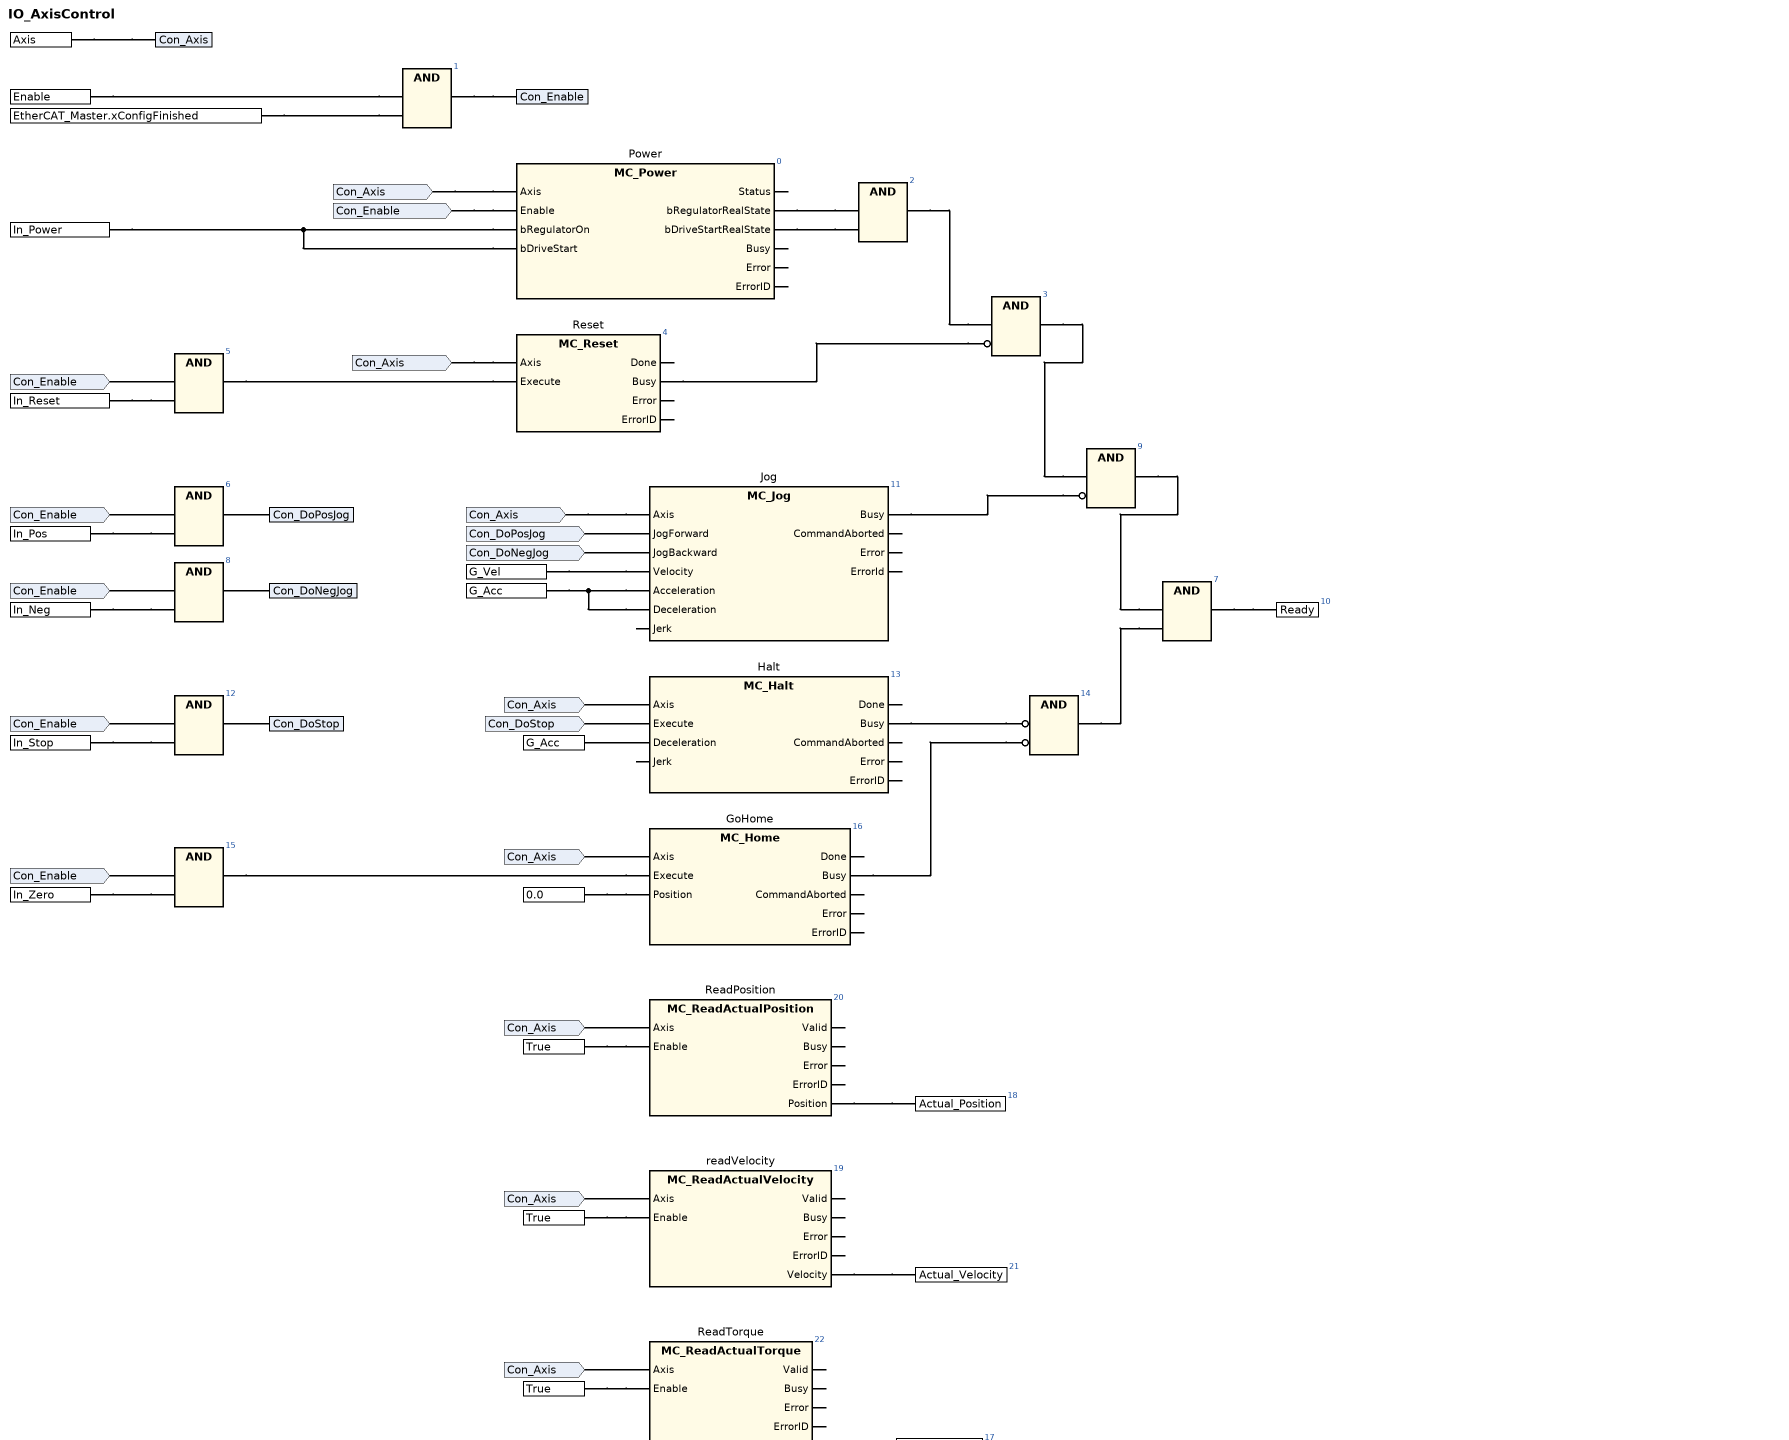
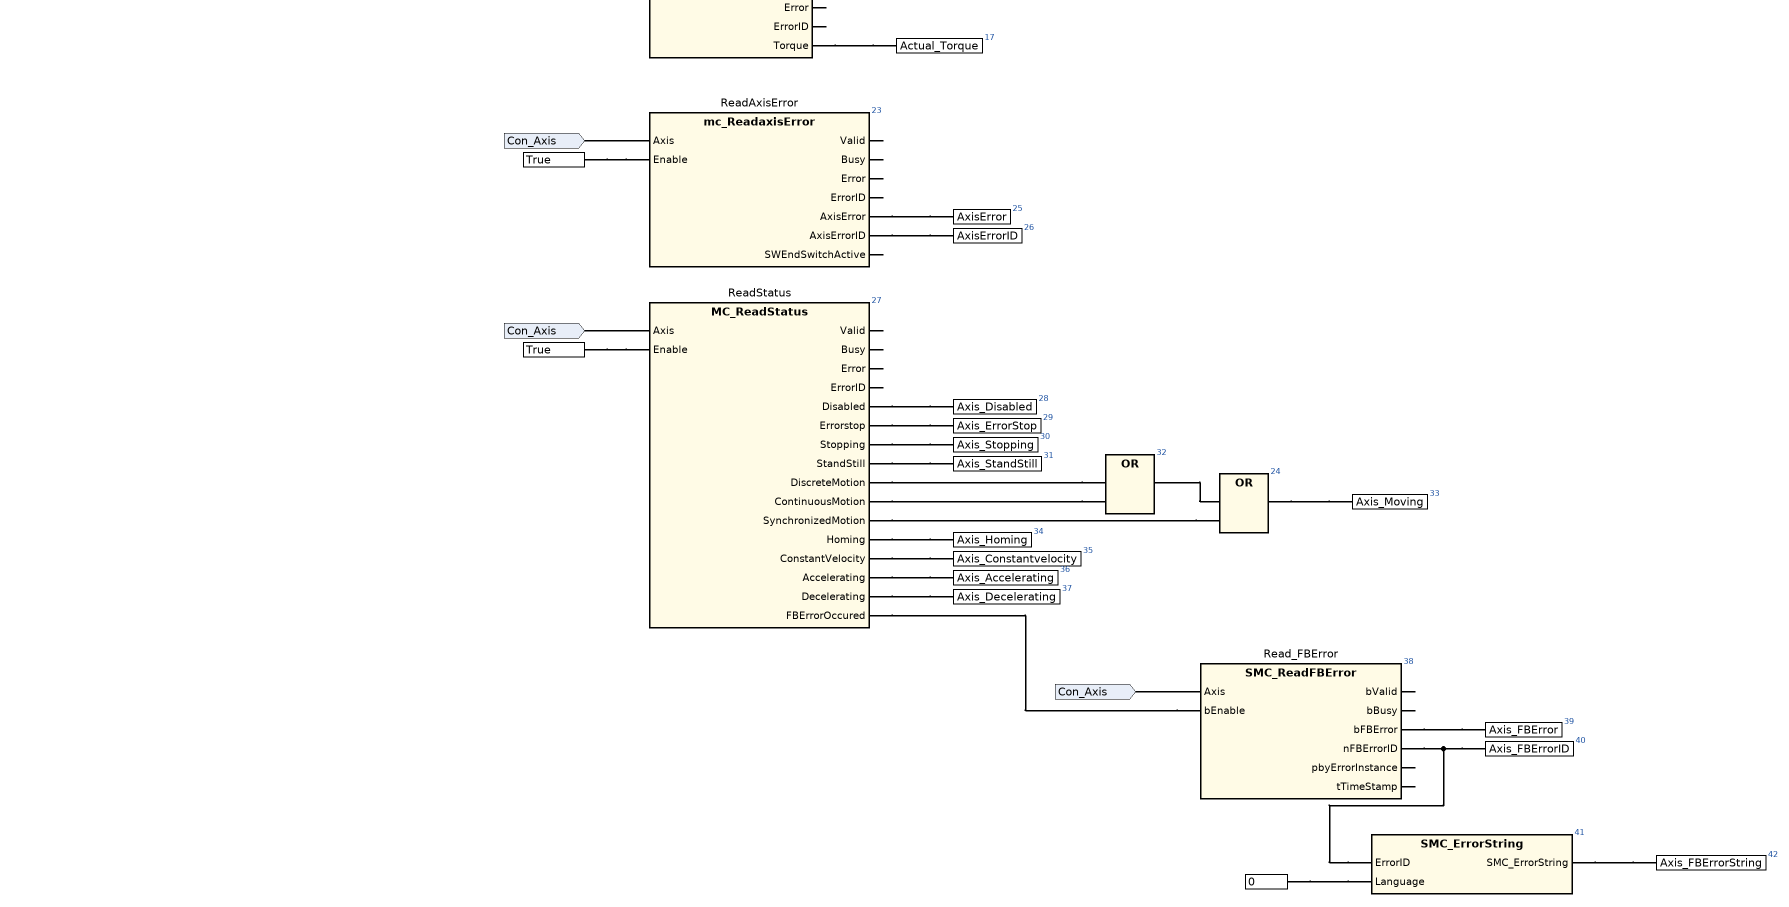
Power(Axis := _w1, Enable := _w2, bRegulatorOn := In_Power, bDriveStart := In_Power); // MC_Power
(* Enable AND EtherCAT_Master.xConfigFinished; result not used *)
_w3 := (Power.bRegulatorRealState AND Power.bDriveStartRealState) AND NOT Reset.Busy;
Reset(Axis := _w4, Execute := _w5); // MC_Reset
_w5 := _w6 AND In_Reset;
(* _w7 AND In_Pos; result not used *)
_w10 := _w8 AND _w9;
(* _w11 AND In_Neg; result not used *)
_w8 := _w3 AND NOT Jog.Busy;
Ready := _w10;
Jog(
    Axis := _w12,
    JogForward := _w13,
    JogBackward := _w14,
    Velocity := G_Vel,
    Acceleration := G_Acc,
    Deceleration := G_Acc); // MC_Jog
(* _w15 AND In_Stop; result not used *)
Halt(Axis := _w16, Execute := _w17, Deceleration := G_Acc); // MC_Halt
_w9 := NOT Halt.Busy AND NOT GoHome.Busy;
GoHome(Axis := _w19, Execute := _w18 AND In_Zero, Position := 0.0); // MC_Home
Actual_Torque := ReadTorque.Torque;
Actual_Position := ReadPosition.Position;
readVelocity(Axis := _w20, Enable := True); // MC_ReadActualVelocity
ReadPosition(Axis := _w21, Enable := True); // MC_ReadActualPosition
Actual_Velocity := readVelocity.Velocity;
ReadTorque(Axis := _w22, Enable := True); // MC_ReadActualTorque
ReadAxisError(Axis := _w23, Enable := True); // mc_ReadaxisError
_w25 := _w24 OR ReadStatus.SynchronizedMotion;
AxisError := ReadAxisError.AxisError;
AxisErrorID := ReadAxisError.AxisErrorID;
ReadStatus(Axis := _w26, Enable := True); // MC_ReadStatus
Axis_Disabled := ReadStatus.Disabled;
Axis_ErrorStop := ReadStatus.Errorstop;
Axis_Stopping := ReadStatus.Stopping;
Axis_StandStill := ReadStatus.StandStill;
_w24 := ReadStatus.DiscreteMotion OR ReadStatus.ContinuousMotion;
Axis_Moving := _w25;
Axis_Homing := ReadStatus.Homing;
Axis_Constantvelocity := ReadStatus.ConstantVelocity;
Axis_Accelerating := ReadStatus.Accelerating;
Axis_Decelerating := ReadStatus.Decelerating;
Read_FBError(Axis := _w27, bEnable := ReadStatus.FBErrorOccured); // SMC_ReadFBError
Axis_FBError := Read_FBError.bFBError;
Axis_FBErrorID := Read_FBError.nFBErrorID;
_w28 := SMC_ErrorString(ErrorID := Read_FBError.nFBErrorID, Language := 0);
Axis_FBErrorString := _w28;

END_FUNCTION_BLOCK

// LogHiCycleCount
PROGRAM LogHiCycleCount
VAR
	strMsg: STRING[255];
	iStatus : INT := 0;
	LogIndex :DINT := 0;
	LogMsg : ARRAY [1..200] OF STRING[255];
	LogType : STRING;
	
	CycleTimeWarning: DWORD := 600;
	TotalSyncBufferAvgWarning: DINT := 125;
	CycleTimeError: DWORD := 900;
	TotalSyncBufferAvgError: DINT := 200;
END_VAR

VAR_INPUT
	bResetArray: BOOL;
END_VAR


IF bResetArray = TRUE THEN
	LogIndex := 0;
END_IF




CASE iStatus OF
	
0:	//Wait for Distributed Clocks in sync
	IF GVL.DC_InSync THEN
		iStatus:=iStatus + 1;
	END_IF
1: 	//Wait for High Cycle Count
	LogType := 'None';
	IF (DC_Monitor.CycleTime_Last > CycleTimeWarning OR DC_Monitor.TotalSyncBufferAvg > TotalSyncBufferAvgWarning) THEN
		iStatus := iStatus + 1;
	END_IF

2:	//Log Data
	LogIndex := LogIndex + 1;
	IF (DC_Monitor.CycleTime_Last > CycleTimeError OR DC_Monitor.TotalSyncBufferAvg > TotalSyncBufferAvgError) THEN
		LogType := 'Error';
	ELSE
		LogType := 'Warning';
	END_IF
	LogMsg[LogIndex] :=  GetLogMsgString();
	
	iStatus := 2;

END_CASE

END_PROGRAM

// GetLogMsgString
FUNCTION GetLogMsgString : STRING[255]
VAR_INPUT
END_VAR
VAR
	msg: STRING[255];
	seperator: STRING;
	eol:String;
	
	strTemp0: STRING[255];
	strTemp1: STRING[255];
END_VAR

eol := WORD_AS_STRING(16#0A0D, FALSE);
seperator := ',';

(*
strTemp0 := Concat(Concat(Concat(Concat(Concat(Concat(Concat(Concat(Concat(Concat(Concat(Concat(Concat(Concat(	My_FLOAT_TO_STRING(X.fSetPosition), 
																												seperator), 
																												My_FLOAT_TO_STRING(Y.fSetPosition)),  
																												seperator), 
																												My_FLOAT_TO_STRING(Z.fSetPosition)),  
																												seperator), 
																												My_FLOAT_TO_STRING(BB.fSetPosition)),  
																												seperator), 
																												My_FLOAT_TO_STRING(CC.fSetPosition)),  
																												seperator), 
																												My_FLOAT_TO_STRING(GGX.fSetPosition)),  
																												seperator), 
																												My_FLOAT_TO_STRING(GGZ.fSetPosition)),  
																												seperator), 
																												My_FLOAT_TO_STRING(GGC.fSetPosition));
																												
strTemp1 := Concat(Concat(Concat(Concat(Concat(Concat(Concat(Concat(Concat(Concat(Concat(Concat(Concat(Concat(	My_FLOAT_TO_STRING(X.fActPosition), 
																												seperator), 
																												My_FLOAT_TO_STRING(Y.fActPosition)),  
																												seperator), 
																												My_FLOAT_TO_STRING(Z.fActPosition)),  
																												seperator), 
																												My_FLOAT_TO_STRING(BB.fActPosition)),  
																												seperator), 
																												My_FLOAT_TO_STRING(CC.fActPosition)),  
																												seperator), 
																												My_FLOAT_TO_STRING(GGX.fActPosition)),  
																												seperator), 
																												My_FLOAT_TO_STRING(GGZ.fActPosition)),  
																												seperator), 
																												My_FLOAT_TO_STRING(GGC.fActPosition));
*)


strTemp0 := My_FLOAT_TO_STRING();
strTemp1 := 'TotalSyncBufferAvg';
GetLogMsgString := Concat(Concat(Concat(Concat(Concat(	GetTimeStampString(),
														seperator),
														strTemp0), 
														seperator),
														strTemp1), 
														eol);

END_FUNCTION

// My_FLOAT_TO_STRING
FUNCTION My_FLOAT_TO_STRING : STRING(10)
VAR_INPUT
	Value : LREAL;
END_VAR
VAR
	intTemp : DINT;
END_VAR

//My_LREAL_TO_STRING := REAL_TO_STRING(Value);
intTemp := LREAL_TO_DINT(Value * 1000);
My_FLOAT_TO_STRING := LREAL_TO_STRING(DINT_TO_LREAL(intTemp)/1000 );

END_FUNCTION

// GetTimeStampString
FUNCTION GetTimeStampString : String
VAR_INPUT
END_VAR
VAR
	TimeStamp : SysTime;
	StructTimeStamp : SysTimeDate;
	Result : RTS_IEC_RESULT;
	StrDate : STRING;
	StrTime : STRING;
	
END_VAR

Result := systimertc.SysTimeRtcHighResGet(pTimestamp := TimeStamp);

Result := systimertc.SysTimeRtcConvertHighResToLocal(pTimeStamp:=TimeStamp, pDate:=StructTimeStamp);

StrDate := UINT_TO_STRING(StructTimeStamp.wYear);
IF StructTimeStamp.wMonth < 10 THEN 
	StrDate := Concat(Concat(StrDate, '0') , UINT_TO_STRING(StructTimeStamp.wMonth));
ELSE
	StrDate := Concat(StrDate , UINT_TO_STRING(StructTimeStamp.wMonth));
END_IF

IF StructTimeStamp.wDay < 10 THEN 
	StrDate := Concat(Concat(StrDate , '0') , UINT_TO_STRING(StructTimeStamp.wDay));
ELSE
	StrDate := Concat(StrDate , UINT_TO_STRING(StructTimeStamp.wDay));
END_IF


IF StructTimeStamp.wHour < 10 THEN 
	StrTime := Concat(Concat('0' , UINT_TO_STRING(StructTimeStamp.wHour)) , ':');
ELSE
	StrTime := Concat(UINT_TO_STRING(StructTimeStamp.wHour) , ':');
END_IF

IF StructTimeStamp.wMinute < 10 THEN 
	StrTime := Concat(Concat(Concat(StrTime , '0') , UINT_TO_STRING(StructTimeStamp.wMinute)), ':');
ELSE
	StrTime := Concat(Concat(StrTime , UINT_TO_STRING(StructTimeStamp.wMinute)), ':');
END_IF

IF StructTimeStamp.wSecond < 10 THEN 
	StrTime := Concat(Concat(Concat(StrTime , '0') , UINT_TO_STRING(StructTimeStamp.wSecond)) , '.');
ELSE
	StrTime := Concat(Concat(StrTime , UINT_TO_STRING(StructTimeStamp.wSecond)) , '.');
END_IF

IF StructTimeStamp.wMilliseconds < 10 THEN 
	StrTime := Concat(Concat(StrTime , '00') , UINT_TO_STRING(StructTimeStamp.wMilliseconds));
ELSE
	IF StructTimeStamp.wMilliseconds < 100 THEN 
		StrTime := Concat(Concat(StrTime , '0') , UINT_TO_STRING(StructTimeStamp.wMilliseconds));
	ELSE
		StrTime := Concat(StrTime , UINT_TO_STRING(StructTimeStamp.wMilliseconds));
	END_IF
END_IF

//GetTimeStampString := Concat(Concat(strDate , '-'), strTime);
GetTimeStampString := strTime;

END_FUNCTION

// PLC_PRG_1
PROGRAM PLC_PRG_1
VAR
	(* Regression Test Alarms 4.0 *)
    SLCTag: INT;
	SLCTag2: INT;
	Ramp1: INT;
	
	(* Regresstion Test Comparison Test 4.0 *)
	SimBool1 : BOOL;
	SimBool2 : BOOL;
	SimBool3 : BOOL;
	SimInt1 : INT;
	SimInt2: INT;
	SimString1 : STRING;
	SimString2 : STRING;
	
	(* Regression Test Connections Test 4.0 *)
	Ramp2: INT;
	
	(* Regression Test Data Type Test 4.0 *)
	SimDint1 : DINT;
	SimReal1 : REAL;
	SimLReal1 : LREAL;
	SimSint1 : SINT;
	SimUDint1 : UDINT;
	SimUInt1 : UINT;
	SimUSint1 : USINT;
	
	(* Regression Test Functions and Operators *)
	Ramp3: INT;
	Ramp4: INT;
	Ramp5: INT;
	Ramp6: INT;
	Ramp7: INT;
	Ramp8: REAL;
	Ramp10: REAL;
	Ramp11: REAL;
	Ramp12: REAL;
	Ramp13: REAL;
	Ramp14: REAL;
	Ramp15: REAL;
	Ramp16: REAL;
	Ramp17: REAL;
	Ramp18: REAL;
	Ramp19: REAL;
	Ramp20: REAL;
	Ramp9: INT;
	
	Ramp21: DINT;
	Ramp22: DINT;
	Ramp23: DINT;
	Ramp24: DINT;
	Ramp25: DINT;
	Ramp26: DINT;
    Ramp27: DINT;
    Ramp28: DINT;
	Ramp29: DINT;
	Ramp30: DINT;
	Ramp31: DINT;
	Ramp32: DINT;
	Ramp33: DINT;
	Ramp34: DINT;
	Ramp35: DINT;
	Ramp36: DINT;
	Ramp37: DINT;
	Ramp38: DINT;
	Ramp39: DINT;
	Ramp40: DINT;
	Ramp41: DINT;
	Ramp42: DINT;
	Ramp43: DINT;
	Ramp44: DINT;
	Ramp45: DINT;
	Ramp46: DINT;
	Ramp47: DINT;
	Ramp48: DINT;
	Ramp49: DINT;
	Ramp50: DINT;

	RampSTRING: STRING;
	RampSTRINGDummy: INT;
	
	(* Regresstion Test Language Translation *)
	IndicatorRamp1 :INT;
	IndicatorRamp2 :INT;
	IndicatorRamp3 :INT;
	MessageTableRamp :INT;
	RangeIndicatorRamp :INT;
	
	(* Regression Test Styles *)
	StylesRamp :INT;
	
	(* Regression Test Summing *)
	SimTag1DefaultInitial :INT;
	SimTag1IntInitial :INT;
	SimTag2DefaultInitial :INT;
	SimTag2IntInitial :INT;
	
	(* Regression Test System Tags *)
	DeviceDay :UINT;
	DeviceHour :UINT;
	DeviceMinute :UINT;
	DeviceMonth :UINT;
	DeviceSecond :UINT;
	DeviceYear :UINT;
		
	MyCounter: INT; (* 1000ms *)
	MyCounter1: INT;
	MyCounter2: INT;
	MyCounter3: INT; (* 2000ms *)
	MyCounter4: INT;
	MyCounter5: INT; (* 500ms *)
	MyCounter6: INT; (* 250ms *)
END_VAR

(* Regression Test Alarms 4.0 *)
  MyCounter := MyCounter + 1;
    IF MyCounter = 4 THEN
		Ramp1 := Ramp1 + 1;
		Ramp2 := Ramp2 + 1;
		IndicatorRamp2 := IndicatorRamp2 + 1;
		MessageTableRamp := MessageTableRamp + 1;
		IF Ramp1 = 6 THEN
			Ramp1 := 1;
		END_IF
		IF Ramp2 = 101 THEN
			Ramp2 := 1;
		END_IF
		IF IndicatorRamp2 = 2 THEN
			IndicatorRamp2 := 0;
		END_IF
		IF MessageTableRamp = 4 THEN
			MessageTableRamp :=1;
		END_IF
		MyCounter :=0;
	END_IF
	
(* Regression Test Functions and Operators *)
  MyCounter1 := MyCounter1 + 1;
  IF MyCounter1 = 4 THEN
	 Ramp3 := Ramp3 + 1;
     Ramp5 := Ramp5 + 1;
	 Ramp9 := Ramp9 + 1;
     IF Ramp3 = 11 THEN
		 Ramp3 :=0;
	 END_IF
	 IF Ramp5 = 2 THEN
		 Ramp5 :=0;
	 END_IF
	 IF Ramp9 = 11 THEN
		 Ramp9 := -10;	 
	 END_IF
	 MyCounter1 := 0;
  END_IF
  
  MyCounter2 := MyCounter2 + 1;
  IF MyCounter2 = 6 THEN
	 Ramp4 := Ramp4 + 1;
     Ramp6 := Ramp6 + 1;
     IF Ramp4 = 11 THEN
		 Ramp4 :=0;
	 END_IF
	 IF Ramp6 = 2 THEN
		 Ramp6 :=0;
	 END_IF
	 MyCounter2 := 0;
  END_IF
  
  MyCounter3 := MyCounter3 + 1;
  IF MyCounter3 = 8 THEN
	 Ramp7 := Ramp7 + 1;
     Ramp8 := Ramp8 + 0.1;
	 Ramp10 := Ramp10 + 0.21;
	 Ramp11 := Ramp11 + 0.211;
	 Ramp12 := Ramp12 + 0.32;
	 Ramp13 := Ramp13 + 0.43;
	 Ramp14 := Ramp14 + 0.561;
	 Ramp15 := Ramp15 + 0.78;
	 Ramp16 := Ramp16 + 0.902;
	 Ramp17 := Ramp17 + 0.704;
	 Ramp18 := Ramp18 + 0.2222;
	 Ramp19 := Ramp19 + 0.111;
	 Ramp20 := Ramp20 + 0.2211;
	 IndicatorRamp3 := IndicatorRamp3 + 1;
     IF Ramp7 = 361 THEN
		 Ramp7 :=0;
	 END_IF
	 IF Ramp8 >= 1 THEN
		 Ramp8 :=0;
		 Ramp10 :=0;
		 Ramp11 :=0;
		 Ramp12 :=0;
		 Ramp13 :=0;
		 Ramp14 :=0;
		 Ramp15 :=0;
		 Ramp16 :=0;
		 Ramp17 :=0;
		 Ramp18 :=0;
		 Ramp19 :=0;
		 Ramp20 :=0;
	 END_IF
	 IF IndicatorRamp3 = 2 THEN
		 IndicatorRamp3 :=0;
	 END_IF
	 MyCounter3 :=0;
  END_IF
  
  MyCounter4 := MyCounter4 + 1;
  IF MyCounter4 = 4 THEN
	  RampSTRINGDummy := RampSTRINGDummy + 1;
	  IF RampSTRINGDummy = 1 THEN
		  RampSTRING := 'Parker Hannifin';
	  END_IF
	  IF RampSTRINGDummy = 2 THEN
		  RampSTRING := 'TestMessage';
		  RampSTRINGDummy := 0;
	  END_IF
	  MyCounter4 := 0;
  END_IF
  
  (* Regression Test Language Translation *)
  MyCounter5 := MyCounter5 + 1;
  IF MyCounter5 = 2 THEN
	  IndicatorRamp1 := IndicatorRamp1 + 1;
	  IF IndicatorRamp1 = 2 THEN
		  IndicatorRamp1 := 0;
	  END_IF
	  MyCounter5 :=0;
  END_IF
  
  RangeIndicatorRamp := RangeIndicatorRamp + 1;
  IF RangeIndicatorRamp = 61 THEN
	  RangeIndicatorRamp :=1;
  END_IF
  
  (* Regression Test Styles *)
  MyCounter6 := MyCounter6 + 1;
  IF MyCounter6 = 1 THEN
	  StylesRamp := StylesRamp + 1;
	  IF StylesRamp = 101 THEN
		  StylesRamp := 0;
	  END_IF
	  MyCounter6 :=0;
  END_IF
  
  Ramp21 := Ramp21 + 1;
  Ramp22 := Ramp22 + 1;
  Ramp23 := Ramp23 + 1;
  Ramp24 := Ramp24 + 1;
  Ramp25 := Ramp25 + 1;
  Ramp26 := Ramp26 + 1;
  Ramp27 := Ramp27 + 1;
  Ramp28 := Ramp28 + 1;
  Ramp29 := Ramp29 + 1;
  Ramp30 := Ramp30 + 1;
  Ramp31 := Ramp31 + 1;
  Ramp32 := Ramp32 + 1;
  Ramp33 := Ramp33 + 1;
  Ramp34 := Ramp34 + 1;
  Ramp35 := Ramp35 + 1;
  Ramp36 := Ramp36 + 1;
  Ramp37 := Ramp37 + 1;
  Ramp38 := Ramp38 + 1;
  Ramp39 := Ramp39 + 1;
  Ramp40 := Ramp40 + 1;
  Ramp41 := Ramp41 + 1;
  Ramp42 := Ramp42 + 1;
  Ramp43 := Ramp43 + 1;
  Ramp44 := Ramp44 + 1;
  Ramp45 := Ramp45 + 1;
  Ramp46 := Ramp46 + 1;
  Ramp47 := Ramp47 + 1;
  Ramp48 := Ramp48 + 1;
  Ramp49 := Ramp49 + 1;
  Ramp50 := Ramp50 + 1;
  IF Ramp21 > 200000000 THEN
	  Ramp21:=0;
	  Ramp22:=0;
	  Ramp23:=0;
	  Ramp24:=0;
	  Ramp25:=0;
	  Ramp26:=0;
	  Ramp27:=0;
	  Ramp28:=0;
	  Ramp29:=0;
	  Ramp30:=0;
	  Ramp31:=0;
	  Ramp32:=0;
	  Ramp33:=0;
	  Ramp34:=0;
	  Ramp35:=0;
	  Ramp36:=0;
	  Ramp37:=0;
	  Ramp38:=0;
	  Ramp39:=0;
	  Ramp40:=0;
	  Ramp41:=0;
	  Ramp42:=0;
	  Ramp43:=0;
	  Ramp44:=0;
	  Ramp45:=0;
	  Ramp46:=0;
	  Ramp47:=0;
	  Ramp48:=0;
	  Ramp49:=0;
	  Ramp50:=0;
  END_IF

END_PROGRAM

// Run_FileCopy
PROGRAM Run_FileCopy
VAR
	RunTest: Test_FileCopy;
END_VAR

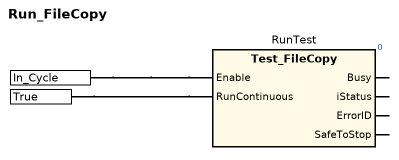
RunTest(Enable := In_Cycle, RunContinuous := True); // Test_FileCopy

END_PROGRAM

// Test_FileCopy
FUNCTION_BLOCK Test_FileCopy
VAR_INPUT
	Enable: BOOL;
	RunContinuous:Bool := False;
END_VAR
VAR_OUTPUT
	Busy: BOOL;
	iStatus : INT := 0;
	ErrorID: INT;
	SafeToStop : Bool;
END_VAR
VAR
	OriginalFilePath : STRING := '/Hard disk/Backup/nk.bin';
	MemoryFilePath : STRING := '/nk.bin';
	USBFilePath : STRING := '/Hard disk2/nk.bin';
	DwellTime : TIME := T#15S;
	DoDwell : TON;
	
	Result1: SYSFILE.RTS_IEC_RESULT;
	Result2: SYSFILE.RTS_IEC_RESULT;

	BytesCopied: DWORD;
	SizeOriginal: DWORD;
	SizeMemory: DWORD;
	SizeUSB: DWORD;
END_VAR

IF Enable = FALSE and SafeToStop = True THEN
	iStatus := 0;
END_IF


CASE iStatus OF
	
0:	//Wait for Distributed Clocks in sync
	SafeToStop:=TRUE;
	IF Enable:= TRUE AND EtherCAT_Master.xConfigFinished AND DC_InSync THEN
		Busy:=TRUE;
		ErrorID:=0;
		iStatus:=iStatus + 1;
	END_IF
1: //Check Original File Exist
	SafeToStop:=TRUE;
	SizeOriginal := SysFileGetSize(OriginalFilePath, ADR(Result1));
	IF SizeOriginal > 0 AND Result1 = Errors.ERR_OK THEN
		iStatus:=iStatus + 1;
	ELSE
		ErrorID := -1 * iStatus;  //Original does not exist
		iStatus := 99;
	END_IF
2:	//Delete Copy in Memory
	SafeToStop:=FALSE;
	SizeMemory := SysFileGetSize(MemoryFilePath, ADR(Result1));
	IF Result1 = Errors.ERR_NO_OBJECT THEN	
		iStatus:=iStatus + 1;
	ELSE
		Result1 := SysFileDelete(MemoryFilePath);
		IF Result1 = Errors.ERR_OK THEN
			iStatus:=iStatus + 1;
		ELSE
			ErrorID := -1 * iStatus;  //Delete Memory Copy Failed
			iStatus := 99;
		END_IF
	END_IF
		
3:	//Delete Copy on USB Thumbdrive
	SafeToStop:=FALSE;
	SizeUSB := SysFileGetSize(USBFilePath, ADR(Result1));
	IF Result1 = Errors.ERR_NO_OBJECT THEN
		iStatus:=iStatus + 1;
	ELSE
		Result1 := SysFileDelete(USBFilePath);
		IF Result1 = Errors.ERR_OK THEN
			iStatus:=iStatus + 1;
		ELSE
			ErrorID := -1 * iStatus;  //Delete USB Copy Failed
			iStatus := 99;
		END_IF
	END_IF
	
4:  //Do Initial Dwell
	SafeToStop:=TRUE;
	DoDwell(PT:=DwellTime, IN:=TRUE);
	IF DoDwell.Q = TRUE THEN
		DoDwell(PT:=DwellTime, IN:=FALSE);
		iStatus:=iStatus + 1;
	END_IF

5:	// Copy to Memory 
	SafeToStop:=FALSE;
	Result1:=SysFileCopy(MemoryFilePath,OriginalFilePath, ADR(BytesCopied));
	IF Result1=Errors.ERR_OK AND BytesCopied=SizeOriginal THEN
		iStatus:=iStatus + 1;
	ELSE
		ErrorID := -1 * iStatus;  //Copy to Memory Failed
		iStatus := 99;
	END_IF
	
6:	//Do Initial Dwell
	SafeToStop:=TRUE;
	DoDwell(PT:=DwellTime, IN:=TRUE);
	IF DoDwell.Q = TRUE THEN
		DoDwell(PT:=DwellTime, IN:=FALSE);
		iStatus:=iStatus + 1;
	END_IF

7:  // Copy to USBThumbdrive 
	SafeToStop:=FALSE;
	Result1:=SysFileCopy(USBFilePath,OriginalFilePath, ADR(BytesCopied));
	IF Result1=Errors.ERR_OK AND BytesCopied=SizeOriginal THEN
		iStatus:=iStatus + 1;
	ELSE
		ErrorID := -1 * iStatus;  //Copy to Memory Failed
		iStatus := 99;
	END_IF
	
8:	//Do Initial Dwell
	SafeToStop:=TRUE;
	DoDwell(PT:=DwellTime, IN:=TRUE);
	IF DoDwell.Q = TRUE THEN
		DoDwell(PT:=DwellTime, IN:=FALSE);
		iStatus:=iStatus + 1;
	END_IF

9:  //Check Memory File Exist
	SafeToStop:=TRUE;
	SizeMemory := SysFileGetSize(MemoryFilePath, ADR(Result1));
	IF SizeMemory > 0 AND Result1 = Errors.ERR_OK THEN
		iStatus:=iStatus + 1;
	ELSE
		ErrorID := -1 * iStatus;  //Memory does not exist
		iStatus := 99;
	END_IF	

10:  //Check USB File Exist
	SafeToStop:=TRUE;
	SizeUSB := SysFileGetSize(USBFilePath, ADR(Result1));
	IF SizeUSB > 0 AND Result1 = Errors.ERR_OK THEN
		IF RunContinuous=TRUE THEN
			iStatus:=0;
		ELSE
			iStatus := 99;
		END_IF	
	ELSE
		ErrorID := -1 * iStatus;  //USB does not exist
		iStatus := 99;
	END_IF	
	


99: //Got Error
	SafeToStop:=TRUE;
	Busy:=FALSE;
	
END_CASE

	B_Output07:= SafeToStop;
	B_Output06:= SafeToStop;
	B_Output05:= SafeToStop;
	B_Output04:= SafeToStop;
	B_Output03:= SafeToStop;
	B_Output02:= SafeToStop;
	B_Output01:= SafeToStop;
	B_Output00:= SafeToStop;

END_FUNCTION_BLOCK

// LogData
PROGRAM LogData
VAR
	filename: STRING := '/Windows/Logs/Log_HighCycleCount.csv';
	filehandle: SYSFILE.RTS_IEC_HANDLE;
	strMsg: STRING[255];
	FOResult: SYSFILE.RTS_IEC_RESULT;
	FWResult: SYSFILE.RTS_IEC_RESULT;
	FWStatus: POINTER TO RTS_IEC_RESULT;
	FCResult: SYSFILE.RTS_IEC_RESULT;
	bytesWritten: DWORD;
	bFileOpen: BOOL;
	iStatus : INT := 0;
	
	
	SafeToStop: BOOL;
	Result1: SYSFILE.RTS_IEC_RESULT;
	SizeFile: DWORD;
	ErrorID: INT;
	diActPosition: UDINT;
	
	LogIndex :DINT := 0;
	LogMsg : ARRAY [1..200] OF STRING[255];
	LogType : STRING;

	intIndex: DINT;
END_VAR






CASE iStatus OF
	
0:	//Wait for Distributed Clocks in sync
	SafeToStop:=TRUE;
	IF EtherCAT_Master.xConfigFinished THEN
		iStatus:=iStatus + 1;
	END_IF
1: 	//Delete Copy in Memory
	SafeToStop:=FALSE;
	SizeFile := SysFileGetSize(filename, ADR(Result1));
	IF Result1 = Errors.ERR_NO_OBJECT THEN	
		iStatus:=iStatus + 1;
	ELSE
		Result1 := SysFileDelete(filename);
		IF Result1 = Errors.ERR_OK THEN
			iStatus:=iStatus + 1;
		ELSE
			ErrorID := -1 * iStatus;  //Delete Memory Copy Failed
			iStatus := 99;
		END_IF
	END_IF

2: 	//Open File
	filehandle := SysFileOpen(szFile := filename, am := AM_WRITE, pResult:= ADR(FOResult));
	IF (filehandle <> 16#00000000 AND filehandle <> 16#FFFFFFFF AND FOResult = ERRORS.ERR_OK) THEN 
		bFileOpen := TRUE;
		iStatus := iStatus + 1;
	ELSE
		ErrorID := -1 * iStatus;  //Open Memory Copy Failed
		iStatus := 99;
	END_IF

3:	//Write Header Line
	strMsg := GetHeaderString();
	bytesWritten:= SysFileWrite(filehandle, ADR(strMsg), DINT_TO_DWORD(LEN(strMsg)), ADR(FWResult));
	IF bytesWritten = DINT_TO_DWORD(LEN(strMsg)) THEN
		iStatus := iStatus + 1;
	ELSE
		ErrorID := -1 * iStatus;  //Write Header Failed
		iStatus := 100;
	END_IF

4:  //Close File
	FCResult := SysFileClose(filehandle);
	IF FCResult = ERRORS.ERR_OK THEN
		SafeToStop:=TRUE;
	ELSE
		ErrorID := -1 * iStatus;  //File Close Failed
		iStatus := 99;
	END_IF

5:	// Wait for trigger and Copy Data
	SafeToStop:= TRUE;
	LogHiCycleCount.bResetArray := FALSE;
	LogIndex := LogHiCycleCount.LogIndex;
	IF LogIndex > 0 THEN
		LogMsg := LogHiCycleCount.LogMsg;
	
		LogHiCycleCount.bResetArray := TRUE;
		iStatus:=iStatus + 1;
	END_IF
	

6: //Open File
	
	SafeToStop := FALSE;
	filehandle := SysFileOpen(szFile := filename, am := AM_WRITE, pResult:= ADR(FOResult));
	IF (filehandle <> 16#00000000 AND filehandle <> 16#FFFFFFFF AND FOResult = ERRORS.ERR_OK) THEN 
		bFileOpen := TRUE;
		iStatus := iStatus + 1;
	ELSE
		ErrorID := -1 * iStatus;  //Open Memory Copy Failed
		iStatus := 99;
	END_IF//Open File

7:	//Log Data
	FOR intIndex := 1 TO LogIndex DO
		strMsg := LogMsg[intIndex];
		bytesWritten:= SysFileWrite(filehandle, ADR(strMsg), DINT_TO_DWORD(LEN(strMsg)), ADR(FWResult));
		IF FWResult <> ERRORS.ERR_OK THEN
			ErrorID := -1 * iStatus;  //Log Data Failed
			iStatus := 100;
		END_IF
	END_FOR

8:  //Close File
	FCResult := SysFileClose(filehandle);
	IF FCResult = ERRORS.ERR_OK THEN
		SafeToStop:=TRUE;
		iStatus := 5;
	ELSE
		ErrorID := -1 * iStatus;  //File Close Failed
		iStatus := 99;
	END_IF

99:	//Sit for Error


100://Close File then Sit for Error
	FCResult := SysFileClose(filehandle);
	IF FCResult <> ERRORS.ERR_OK THEN
		SafeToStop:=TRUE;
	END_IF




END_CASE

	B_Output15:= SafeToStop;
	B_Output14:= SafeToStop;
	B_Output13:= SafeToStop;
	B_Output12:= SafeToStop;
	B_Output11:= SafeToStop;
	B_Output10:= SafeToStop;
	B_Output09:= SafeToStop;
	B_Output08:= SafeToStop;

END_PROGRAM

// GetHeaderString
FUNCTION GetHeaderString : STRING[255]
VAR_INPUT
END_VAR
VAR
	msg: STRING[255];
	seperator: STRING;
	eol:String;
	strTemp0 : STRING[255];
	strTemp1 : STRING[255];
	
END_VAR

eol := WORD_AS_STRING(16#0A0D, FALSE);
seperator := ',';
(*
strTemp0 := Concat(Concat(Concat(Concat(Concat(Concat(Concat(Concat(Concat(Concat(Concat(Concat(Concat(Concat(	'PosX', 
																												seperator), 
																												'PosY'),  
																												seperator), 
																												'PosZ'),  
																												seperator), 
																												'PosB'),  
																												seperator), 
																												'PosC'),  
																												seperator), 
																												'PosGX'),  
																												seperator), 
																												'PosGY'),  
																												seperator), 
																												'PosGZ');
strTemp1 := Concat(Concat(Concat(Concat(Concat(Concat(Concat(Concat(Concat(Concat(Concat(Concat(Concat(Concat(	'ActX', 
																												seperator),
																												'ActY'), 
																												seperator),
																												'ActZ'), 
																												seperator),
																												'ActB'), 
																												seperator),
																												'ActC'), 
																												seperator),
																												'ActGX'), 
																												seperator),
																												'ActGY'), 
																												seperator),
																												'ActGZ');
																												
*)


strTemp0 := 'Cycle Time';
strTemp1 := 'TotalSyncBufferAvg';
GetHeaderString := Concat(Concat(Concat(Concat(Concat(	'TimeStamp', 
														seperator),
														strTemp0), 
														seperator),
														strTemp1), 
														eol);

END_FUNCTION

// PLC_PRG
PROGRAM PLC_PRG
VAR
END_VAR

END_PROGRAM

// RunSDO_AOut
PROGRAM RunSDO_AOut
VAR
	iStatus: INT := -1;
	iCycle: INT;
	iCycleMin: INT := -10;
	iCycleMax: INT := 2460;
	DoOutputs : SetSDO_AOut;
	DoInputs : GetSDO_AOut;
	TimerON : TON;
	tWait: TIME := T#500ms;
	iIncrement: INT := 123;
	rExpectedValue: REAL;
	rActualValue: REAL;
//	cavConfig: ConfigAnalogVoltage;
	ResetError: BOOL;
	
	ValueMin1: REAL;
	ValueMax1: REAL;
	ValueMin2: REAL;
	ValueMax2: REAL;
	
	Got_DC_OutOfSync: BOOL;

	ExpectedValue1: INT;
	ExpectedValue2: INT;
	ActualValue1: INT;
	ActualValue2: INT;
	
	AOut1_Passed : BOOL;
	AOut2_Passed : BOOL;
	
END_VAR


IF iStatus > -1 AND NOT(DC_InSync) THEN
	Got_DC_OutOfSync := TRUE;
	iStatus := -100;
END_IF

CASE iStatus OF
-100: //Wait for Recovery to Finish
	DoOutputs(Axis := X, Execute:=FALSE);
	DoInputs(Axis := X, Execute:=FALSE);
	TimerON(IN:=FALSE,PT:=T#0S);
	IF Recovery.InRecovery = FALSE AND Recovery.Done THEN	
		iStatus := -1;
	END_IF;
	
	
-1: //Wait for EtherCAT
	IF EtherCAT_Master.xConfigFinished AND DC_InSync THEN
		iStatus:=iStatus + 1;
	END_IF
	
0: //Set Outputs
	ExpectedValue1 := 0 + iCycle;
	ExpectedValue2 := 0 - iCycle;
	
	DoOutputs(Axis:=X, AOut1 := ExpectedValue1, AOut2 := ExpectedValue2, Execute:=TRUE);
	
	IF DoOutputs.Done THEN
		iCycle:=iCycle + iIncrement;
		IF iCycle >= iCycleMax THEN
			iCycle:=0;
		END_IF;
		iStatus := iStatus + 1;	
	END_IF
1: //Wait Time
	TimerON(PT:=tWait, IN:=TRUE);
	IF TimerON.Q=TRUE THEN
		TimerON(IN:=FALSE,PT:=T#0S);
		iStatus := iStatus + 1;
	END_IF
2: //Check Inputs
	DoInputs(Axis:=X, Execute:=TRUE );
	
	IF DoInputs.Done = TRUE THEN
		ActualValue1:=DoInputs.AOut1;
		ActualValue2:=DoInputs.AOut2;
		
		ValueMin1:=ExpectedValue1 * 0.9;
		ValueMax1:=ExpectedValue1 * 1.1;
	
		ValueMin2:=ExpectedValue2 * 1.1;
		ValueMax2:=ExpectedValue2 * 0.9;
		
		AOut1_Passed := (ActualValue1 > ValueMin1) AND (ActualValue1 < ValueMax1);
		AOut2_Passed := (ActualValue2 > ValueMin2) AND (ActualValue2 < ValueMax2);
		
		iStatus := iStatus + 1;	
		DoOutputs(Axis := X, Execute:=FALSE);
		DoInputs(Axis := X, Execute:=FALSE);
	END_IF
3: //Wait Time
	TimerON(PT:=tWait, IN:=TRUE);
	IF TimerON.Q=TRUE THEN
		TimerON(IN:=FALSE,PT:=T#0S);
		iStatus:=0;
	END_IF
	
	
END_CASE;

END_PROGRAM

// SetSDO_AOut
FUNCTION_BLOCK SetSDO_AOut
VAR_IN_OUT
	Axis : AXIS_REF_ETC_SM3;
END_VAR
VAR_INPUT
	Execute:BOOL;
	AOut1: INT;
	AOut2: INT;
END_VAR
VAR_OUTPUT
	Done:BOOL;
	Busy:BOOL;
	Error: BOOL;
	
END_VAR
VAR
	AOut1_PosIndex:UINT:=8977;	//0x2311;
	AOut1_PosSubIndex:USINT:=0;
	AOut2_PosIndex:UINT:=8980;	//0x2314;
	AOut2_PosSubIndex:USINT:=0;
	
	SDO_Write_C3_AOut1: SMC3_ETC_WriteParameter_CoE;
	SDO_Write_C3_AOut2: SMC3_ETC_WriteParameter_CoE;
END_VAR
VAR // added by the converter: edge detectors and wires of the graphical bodies
    _w1 : ANY;
    _w2, _w3 : BOOL;
END_VAR

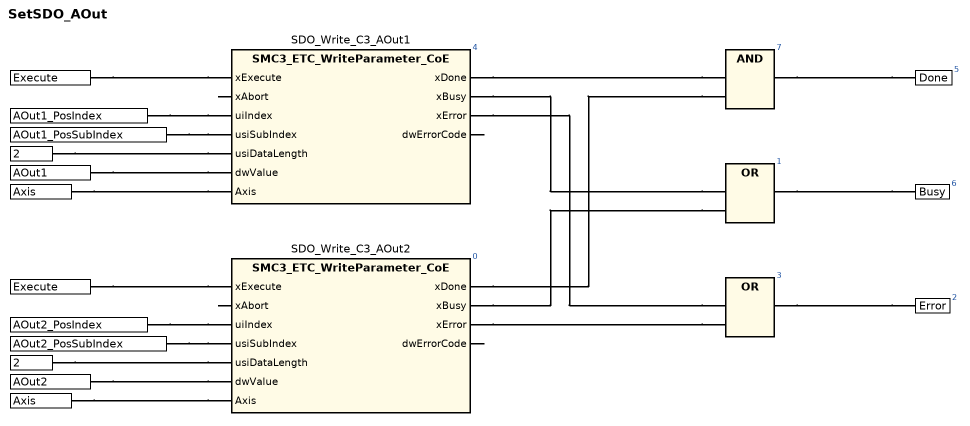
SDO_Write_C3_AOut2(
    xExecute := Execute,
    uiIndex := AOut2_PosIndex,
    usiSubIndex := AOut2_PosSubIndex,
    usiDataLength := 2,
    dwValue := AOut2,
    Axis := Axis); // SMC3_ETC_WriteParameter_CoE
_w1 := SDO_Write_C3_AOut1.xBusy OR SDO_Write_C3_AOut2.xBusy;
Error := _w2;
_w2 := SDO_Write_C3_AOut1.xError OR SDO_Write_C3_AOut2.xError;
SDO_Write_C3_AOut1(
    xExecute := Execute,
    uiIndex := AOut1_PosIndex,
    usiSubIndex := AOut1_PosSubIndex,
    usiDataLength := 2,
    dwValue := AOut1,
    Axis := Axis); // SMC3_ETC_WriteParameter_CoE
Done := _w3;
Busy := _w1;
_w3 := SDO_Write_C3_AOut1.xDone AND SDO_Write_C3_AOut2.xDone;

END_FUNCTION_BLOCK

// GetSDO_AOut
FUNCTION_BLOCK GetSDO_AOut
VAR_IN_OUT
	Axis : AXIS_REF_ETC_SM3;
END_VAR
VAR_INPUT
	Execute:BOOL;
END_VAR
VAR_OUTPUT
	Done:BOOL;
	Busy:BOOL;
	Error: BOOL;
	AOut1: INT;
	AOut2: INT;

END_VAR
VAR
	AOut1_PosIndex:UINT:=8977;	//0x2311;
	AOut1_PosSubIndex:USINT:=0;
	AOut2_PosIndex:UINT:=8980;	//0x2314;
	AOut2_PosSubIndex:USINT:=0;

	SDO_Read_C3_AOut1: SMC3_ETC_ReadParameter_CoE;
	SDO_Read_C3_AOut2: SMC3_ETC_ReadParameter_CoE;
END_VAR
VAR // added by the converter: edge detectors and wires of the graphical bodies
    _w1, _w2, _w3 : BOOL;
    _w4, _w5 : INT;
END_VAR

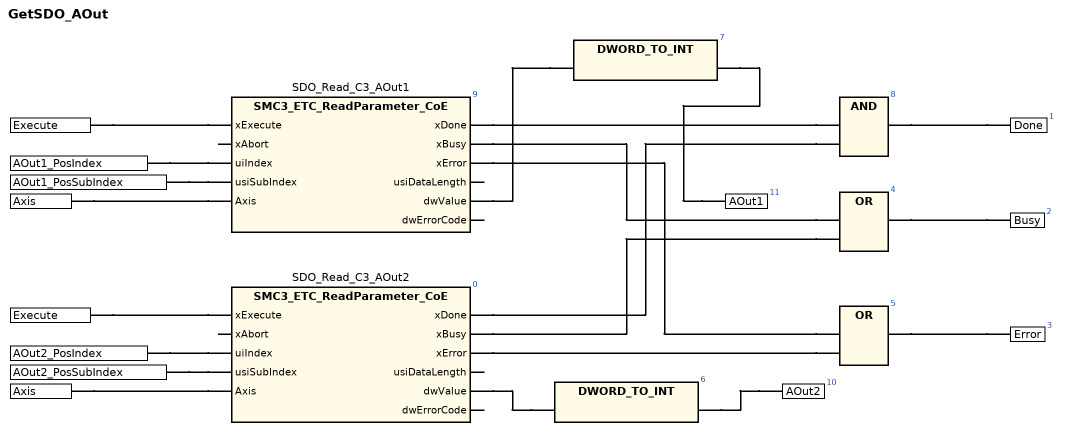
SDO_Read_C3_AOut2(
    xExecute := Execute,
    uiIndex := AOut2_PosIndex,
    usiSubIndex := AOut2_PosSubIndex,
    Axis := Axis); // SMC3_ETC_ReadParameter_CoE
Done := _w1;
Busy := _w2;
Error := _w3;
_w2 := SDO_Read_C3_AOut1.xBusy OR SDO_Read_C3_AOut2.xBusy;
_w3 := SDO_Read_C3_AOut1.xError OR SDO_Read_C3_AOut2.xError;
_w4 := DWORD_TO_INT(SDO_Read_C3_AOut2.dwValue);
_w5 := DWORD_TO_INT(SDO_Read_C3_AOut1.dwValue);
_w1 := SDO_Read_C3_AOut1.xDone AND SDO_Read_C3_AOut2.xDone;
SDO_Read_C3_AOut1(
    xExecute := Execute,
    uiIndex := AOut1_PosIndex,
    usiSubIndex := AOut1_PosSubIndex,
    Axis := Axis); // SMC3_ETC_ReadParameter_CoE
AOut2 := _w4;
AOut1 := _w5;

END_FUNCTION_BLOCK

// ConfigAnalogVoltage
FUNCTION_BLOCK ConfigAnalogVoltage
VAR_INPUT
	Execute: BOOL;
	Channel_Mask: UINT;
END_VAR
VAR_OUTPUT
	Busy: BOOL;
	Done: BOOL;
END_VAR
VAR
	iStatus: INT := 0;
(*	Output00: BOOL;
	Output01: BOOL;
	Output02: BOOL;
	Output03: BOOL;
	Output04: BOOL;
	Output05: BOOL;
	Output06: BOOL;
	Output07: BOOL;
	Output08: BOOL;
	Output09: BOOL;
	Output10: BOOL;
	Output11: BOOL;
	Output12: BOOL;
	Output13: BOOL;
	Output14: BOOL;
	Output15: BOOL;
*)
END_VAR

CASE iStatus OF
	
0: //Waiting for Execute = True
	IF Execute = TRUE THEN
		Busy:=TRUE;
		Done:=FALSE;
		IF Channel_Mask.0 THEN
			AO_Current_Chan0:=FALSE;
			AO_Unipolar_Chan01:=FALSE;
			AO_On_Chan0:=TRUE;
		END_IF
		
		IF Channel_Mask.1 THEN
			AO_Current_Chan1:=FALSE;
			AO_Unipolar_Chan01:=FALSE;
			AO_On_Chan1:=TRUE;
		END_IF
		
		IF Channel_Mask.2 THEN
			AO_Current_Chan2:=FALSE;
			AO_Unipolar_Chan23:=FALSE;
			AO_On_Chan2:=TRUE;
		END_IF
		
		IF Channel_Mask.3 THEN
			AO_Current_Chan3:=FALSE;
			AO_Unipolar_Chan23:=FALSE;
			AO_On_Chan3:=TRUE;
		END_IF
		
		AO_ActiveError0 := TRUE;
		AO_ActiveError1 := TRUE;
		AO_ActiveError2 := TRUE;
		AO_ActiveError3 := TRUE;
		
		
		AI_Unipolar_Chan0 := FALSE;
		AI_Differential_Chan01 := TRUE;
		AI_On_Chan0 := TRUE;
		
		AI_Unipolar_Chan1 := FALSE;
		AI_Differential_Chan23 := TRUE;
		AI_On_Chan1 := TRUE;
		
		AI_Unipolar_Chan2 := FALSE;
		AI_Differential_Chan45 := TRUE;
		AI_On_Chan2 := TRUE;
		
		AI_Unipolar_Chan3 := FALSE;
		AI_Differential_Chan67 := TRUE;
		AI_On_Chan3 := TRUE;
		
		iStatus := iStatus + 1;
		RETURN;
	END_IF;

1:

	AO_SetOptions:=TRUE;
	AI_SetOptions:=TRUE;
	Busy:=FALSE;
	Done:=TRUE;
	iStatus := iStatus + 1;
	RETURN;

2://Waiting for Execute = False
	IF Execute = FALSE THEN
		iStatus := 0;
	END_IF;

END_CASE;

END_FUNCTION_BLOCK

// GetSDO
FUNCTION_BLOCK GetSDO
VAR_IN_OUT
	Axis : AXIS_REF_ETC_SM3;
END_VAR
VAR_INPUT
	Execute:BOOL;
END_VAR
VAR_OUTPUT
	Done:BOOL;
	Busy:BOOL;
	Error: BOOL;
	Position:DWORD;
	
END_VAR
VAR
	SDO_Read_C3_Position: SMC3_ETC_ReadParameter_CoE;
	PosIndex:UINT:=8768; //0x2240
	PosSubIndex:USINT:=0;
END_VAR

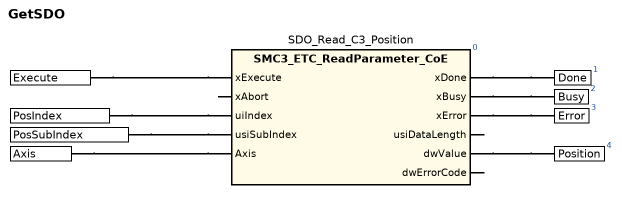
SDO_Read_C3_Position(xExecute := Execute, uiIndex := PosIndex, usiSubIndex := PosSubIndex, Axis := Axis); // SMC3_ETC_ReadParameter_CoE
Done := SDO_Read_C3_Position.xDone;
Busy := SDO_Read_C3_Position.xBusy;
Error := SDO_Read_C3_Position.xError;
Position := SDO_Read_C3_Position.dwValue;

END_FUNCTION_BLOCK

// SetAnalogVoltage
FUNCTION_BLOCK SetAnalogVoltage
VAR_INPUT
	Execute: BOOL;
	Channel_Mask: UINT;
	Channel_0:REAL;
	Channel_1:REAL;
	Channel_2:REAL;
	Channel_3:REAL;
	
END_VAR
VAR_OUTPUT
	Busy: BOOL;
	Done: BOOL;
END_VAR
VAR
	iStatus: INT := 0;
(*	Output00: BOOL;
	Output01: BOOL;
	Output02: BOOL;
	Output03: BOOL;
	Output04: BOOL;
	Output05: BOOL;
	Output06: BOOL;
	Output07: BOOL;
	Output08: BOOL;
	Output09: BOOL;
	Output10: BOOL;
	Output11: BOOL;
	Output12: BOOL;
	Output13: BOOL;
	Output14: BOOL;
	Output15: BOOL;
*)
END_VAR

CASE iStatus OF
	
0: //Waiting for Execute = True
	IF Execute = TRUE THEN
		Busy:=TRUE;
		Done:=FALSE;

		iStatus := iStatus + 1;
		RETURN;
	END_IF;

1:
		IF Channel_Mask.0 THEN
			AO_Chan0:= VOLTS_to_UINT(Channel_0);
		END_IF
		
		IF Channel_Mask.1 THEN
			AO_Chan1:= VOLTS_to_UINT(Channel_1);
		END_IF
		
		IF Channel_Mask.2 THEN
			AO_Chan2:= VOLTS_to_UINT(Channel_2);
		END_IF
		
		IF Channel_Mask.3 THEN
			AO_Chan3:= VOLTS_to_UINT(Channel_3);
		END_IF

	Busy:=FALSE;
	Done:=TRUE;
	iStatus := iStatus + 1;

2://Waiting for Execute = False
	IF Execute = FALSE THEN
		iStatus := 0;
	END_IF;

END_CASE;

END_FUNCTION_BLOCK

// VOLTS_to_UINT
FUNCTION VOLTS_to_UINT : UINT
VAR_INPUT
	Volts:REAL;
END_VAR
VAR
END_VAR

IF Volts > 10 OR Volts < -10 OR Volts = 0.0 THEN //Check out of range or 0
	VOLTS_to_UINT := 0;
ELSE 
	IF Volts > 0 THEN //Case when positive
		VOLTS_to_UINT := REAL_TO_INT(32767 * Volts / 10);
	ELSE //Case when negative
		VOLTS_to_UINT :=  REAL_TO_INT(65535 +(32767 * Volts / 10));
	END_IF
	
END_IF

END_FUNCTION

// UINT_to_VOLTS
FUNCTION UINT_to_VOLTS : REAL
VAR_INPUT
	Counts:UINT;
END_VAR
VAR
END_VAR

IF Counts < 0 OR Counts > 65535 THEN
	UINT_to_VOLTS := 0;
ELSE
	IF Counts <= 32767 THEN
		UINT_to_VOLTS := UINT_TO_REAL(Counts) * 10 / 32767;
	ELSE
		UINT_to_VOLTS := (UINT_TO_REAL(Counts) - 65535) * 10 /32767;	
	END_IF
END_IF

END_FUNCTION

// RunSDO
PROGRAM RunSDO
VAR
	iStatus : INT := -2;
	GetPosition : GetSDO;
	ExpectedValue: REAL;
	ActualValue: DWORD;
	InitializeSDO: InitSDO;
	
	Got_DC_OutOfSync: BOOL;

	InitalValue: DWORD;
END_VAR


IF iStatus > -1 AND NOT(DC_InSync) THEN
	Got_DC_OutOfSync := TRUE;
END_IF

CASE iStatus OF 

-2: //Initialize
	IF EtherCAT_Master.xConfigFinished AND DC_InSync THEN //AND RunMotion.AxisControl.Ready THEN
		InitializeSDO(Axis:= X, Execute:= TRUE);
		GetPosition(Axis:=X, Execute:=TRUE);
		iStatus:=iStatus + 1;
	END_IF

-1: //Wait for Init Finish
	InitializeSDO(Axis:= X, Execute:= TRUE);
	GetPosition(Axis:=X, Execute:=TRUE);
	IF GetPosition.Done THEN
		InitalValue := GetPosition.Position;
		GetPosition(Axis:=X, Execute:=FALSE);
		
		IF InitializeSDO.Done THEN
			InitializeSDO(Axis:= X, Execute:= FALSE);
			iStatus:=iStatus + 1;
		END_IF
	END_IF;
	

0 : //Wait for Dwell
	IF g_MoveDwellPos OR g_MoveDwellNeg THEN
		iStatus:=iStatus + 1;
	END_IF;
	
1 : //Call GetPosition
	GetPosition(Axis:=X, Execute:=TRUE);
	iStatus:=iStatus + 1;
	RETURN;
	
2: //Wait for GetPosition to finish
	GetPosition(Axis:=X, Execute:=TRUE);
	IF GetPosition.Done THEN
		ActualValue := GetPosition.Position;
		GetPosition(Axis:=X, Execute:=FALSE);
		iStatus := iStatus + 1;
	END_IF;
	
3: //Check Position
	IF g_MoveDwellPos THEN
		ExpectedValue := g_PosDistance * 8000 + InitalValue;
		g_GotSDO_PostionPos := ActualValue < (ExpectedValue * 1.1) AND ActualValue > (ExpectedValue *0.9);
	END_IF;
	
	IF g_MoveDwellNeg THEN
		ExpectedValue := g_PosDistance * 4000 + g_NegDistance * 4000 + InitalValue;
		g_GotSDO_PostionNeg := ActualValue < (ExpectedValue * 1.1) AND ActualValue > (ExpectedValue *0.9);
	END_IF;
	iStatus := iStatus + 1;
	
4: //Wait for motion
	IF g_MoveDwellNeg = FALSE AND g_MoveDwellPos = FALSE  THEN
		iStatus := 0;
	END_IF;
	
END_CASE;

END_PROGRAM

// RunMotion
PROGRAM RunMotion
VAR
	AxisControl : IO_AxisControl;
	iStatus: INT := -2;
	DoMove : MC_MoveRelative;
	TimerON:TON;
	tWait : TIME := T#5S;
	tWaitPowerup: TIME := T#30S;
	Got_DC_OutOfSync: BOOL;
	EnableAxisControl: BOOL := FALSE;
	HMI_ActualPosition : INT;
	
	
	

	AxisVar: AXIS_REF_SM3;
	Restart_Axis : SMC3_ReinitDrive;
	TimerRecover : TON;
	ActualPositionX: LREAL;
END_VAR

AxisVar := X;

IF iStatus > -1 AND NOT(DC_InSync) THEN
	Got_DC_OutOfSync := TRUE;
//  Commented out the recovery mechanism to trap the error	
//	iStatus := 10; 
END_IF

CASE iStatus OF
	
-2: //Wait Time
	EnableAxisControl:= FALSE;
	
	//TimerON(PT:=tWaitPowerup, IN:=TRUE);
	IF EtherCAT_Master.xConfigFinished AND DC_InSync THEN
		//TimerON(IN:=FALSE,PT:=T#0S);
		iStatus:=iStatus + 1;
	END_IF
	
-1: //Wait Time
	EnableAxisControl:=TRUE;
	
	IF DC_InSync THEN
		iStatus:=iStatus + 1;
	END_IF
	
	
0: //Wait for Drive to be ready
	//AxisControl(Axis:=X, Enable:=TRUE);
	//In_Power:=TRUE;
	IF AxisControl.Ready AND X.nAxisState=standstill THEN
		IF In_Cycle = TRUE THEN
			iStatus:=iStatus + 1;
		ELSE
			iStatus:=0;	
		END_IF
	END_IF;
	
1: //Start positive move
	DoMove(Axis:=X, Distance:= g_PosDistance, Velocity:=g_Vel, Acceleration:=g_Acc, Deceleration:=g_Acc, Execute:= TRUE);
	IF DoMove.Busy THEN 
		IF In_Cycle = TRUE THEN
			iStatus:=iStatus + 1;
		ELSE
			iStatus:=0;	
		END_IF
	END_IF
	
2: // Wait for Move Finish
	DoMove(Axis:=X, Distance:= g_PosDistance, Velocity:=g_Vel, Acceleration:=g_Acc, Deceleration:=g_Acc, Execute:= TRUE);
	IF DoMove.Done AND X.nAxisState=standstill THEN 
		DoMove(Axis:=X, Execute:= FALSE);
		
		IF In_Cycle = TRUE THEN
			iStatus:=iStatus + 1;
		ELSE
			iStatus:=0;	
		END_IF
	END_IF
	
3: //Wait Time
	g_MoveDwellPos := TRUE;
	TimerON(PT:=tWait, IN:=TRUE);
	IF TimerON.Q=TRUE THEN
		TimerON(IN:=FALSE,PT:=T#0S);
		g_MoveDwellPos :=  FALSE;
		
		IF In_Cycle = TRUE THEN
			iStatus:=iStatus + 1;
		ELSE
			iStatus:=0;	
		END_IF
		
	END_IF

4: //Start negative move
	DoMove(Axis:=X, Distance:= g_NegDistance, Velocity:=g_Vel, Acceleration:=g_Acc, Deceleration:=g_Acc, Execute:= TRUE);
	IF DoMove.Busy THEN 
		IF In_Cycle = TRUE THEN
			iStatus:=iStatus + 1;
		ELSE
			iStatus:=0;	
		END_IF
	END_IF
	
5: // Wait for Move Finish
	DoMove(Axis:=X, Distance:= g_NegDistance, Velocity:=g_Vel, Acceleration:=g_Acc, Deceleration:=g_Acc, Execute:= TRUE);
	IF DoMove.Done AND X.nAxisState=standstill THEN 
		DoMove(Axis:=X, Execute:= FALSE);
		IF In_Cycle = TRUE THEN
			iStatus:=iStatus + 1;
		ELSE
			iStatus:=0;	
		END_IF
	END_IF
	
6: //Wait Time
	g_MoveDwellNeg := TRUE;
	TimerON(PT:=tWait, IN:=TRUE);
	IF TimerON.Q=TRUE THEN
		TimerON(IN:=FALSE,PT:=T#0S);
		g_MoveDwellNeg := FALSE;
		IF In_Cycle = TRUE THEN
			iStatus:= 1;
		ELSE
			iStatus:=0;	
		END_IF
	END_IF

10: //IF DC Out of Sync
	EnableAxisControl:= FALSE;
	EtherCAT_Master.xRestart := TRUE;
	EtherCAT_Master();
	TimerRecover(PT:=tWait, IN:=TRUE);
	IF TimerRecover.Q=TRUE THEN
		TimerRecover(IN:=FALSE,PT:=T#0S);
		iStatus:=11;
	END_IF
	
11: //Re Initialize Drive
	Restart_Axis(Axis:=X, bExecute:= TRUE);
	IF Restart_Axis.bDone THEN
		Restart_Axis(Axis:=X, bExecute:= FALSE);
		g_LostSync := FALSE;
		g_FirstSync := FALSE;
		iStatus := -2;
	END_IF
	
		
END_CASE;

AxisControl(Axis:=X, Enable:=EnableAxisControl);
ActualPositionX:=AxisControl.Actual_Position;
HMI_ActualPosition := LREAL_TO_INT(ActualPositionX * 1000);

END_PROGRAM

// InitSDO
FUNCTION_BLOCK InitSDO
VAR_IN_OUT
	Axis : AXIS_REF_ETC_SM3;
END_VAR
VAR_INPUT
	Execute:BOOL;
END_VAR
VAR_OUTPUT
	Done:BOOL;
	Busy:BOOL;
	Error: BOOL;
	
END_VAR
VAR
	SDOIndex:UINT:=8595;	//0x2193;
	SDOSubIndex:USINT:=0;
	numOutputs : USINT:=3;
	SDO_Write_OutConfig: SMC3_ETC_WriteParameter_CoE;
	iSubIndex: USINT;
END_VAR

numOutputs := 3;

FOR iSubIndex := 1 TO numOutputs DO
	WHILE (NOT(SDO_Write_OutConfig.xDone)) DO
		SDO_Write_OutConfig(uiIndex := SDOIndex, usiSubIndex := iSubIndex, usiDatalength := 2, dwValue := 2, Axis := X, xExecute:= TRUE);	
	END_WHILE;
	SDO_Write_OutConfig(Axis := X, xExecute:= FALSE);
END_FOR;

END_FUNCTION_BLOCK

// GetAnalogVoltage
FUNCTION_BLOCK GetAnalogVoltage
VAR_INPUT
	Execute: BOOL;
	
END_VAR
VAR_OUTPUT
	Busy: BOOL;
	Done: BOOL;
	Channel_0: REAL;
	Channel_1: REAL;
	Channel_2: REAL;
	Channel_3: REAL;
	
END_VAR
VAR
	iStatus: INT := 0;
	
	AI_Chan_0: INT;
	AI_Chan_1: INT;
	AI_Chan_2: INT;
	AI_Chan_3: INT;

	Chan_Raw_0: INT;
	Chan_Raw_1: INT;
	Chan_Raw_2: INT;
	Chan_Raw_3: INT;
	
END_VAR

CASE iStatus OF
	
0: //Waiting for Execute = True
	IF Execute = TRUE THEN
		Busy:=TRUE;
		Done:=FALSE;
		
		
		iStatus := iStatus + 1;
		
	END_IF;

1:	
	Channel_0 := UINT_to_VOLTS(AI_Chan0);
	Channel_1 := UINT_to_VOLTS(AI_Chan1);
	Channel_2 := UINT_to_VOLTS(AI_Chan2);
	Channel_3 := UINT_to_VOLTS(AI_Chan3);
	
	Busy:=FALSE;
	Done:=TRUE;
	iStatus := iStatus + 1;

2://Waiting for Execute = False
	IF Execute = FALSE THEN
		iStatus := 0;
	END_IF;

END_CASE;

END_FUNCTION_BLOCK

// RunMotion_old
PROGRAM RunMotion_old
VAR
	AxisControl : IO_AxisControl;
	iStatus: INT := -2;
	DoMove : MC_MoveRelative;
	TimerON:TON;
	tWait : TIME := T#5S;
	tWaitPowerup: TIME := T#30S;
	Got_DC_OutOfSync: BOOL;

	AxisVar: AXIS_REF_SM3;
	Restart_Axis : SMC3_ReinitDrive;
	TimerRecover : TON;
END_VAR

AxisVar := X;

IF iStatus > -1 AND NOT(DC_InSync) THEN
	Got_DC_OutOfSync := TRUE;
	iStatus := 10;
END_IF

CASE iStatus OF
	
-2: //Wait Time
	//TimerON(PT:=tWaitPowerup, IN:=TRUE);
	IF EtherCAT_Master.xConfigFinished AND DC_InSync THEN
		//TimerON(IN:=FALSE,PT:=T#0S);
		iStatus:=iStatus + 1;
	END_IF
	
-1: //Wait Time
	AxisControl(Axis:=X, Enable:=TRUE);
	IF DC_InSync THEN
		iStatus:=iStatus + 1;
	END_IF
	
	
0: //Wait for Drive to be ready
	AxisControl(Axis:=X, Enable:=TRUE);
	In_Power:=TRUE;
	IF AxisControl.Ready AND X.nAxisState=standstill THEN
		iStatus:=iStatus + 1;	
	END_IF;
	
1: //Start positive move
	DoMove(Axis:=X, Distance:= g_PosDistance, Velocity:=g_Vel, Acceleration:=g_Acc, Deceleration:=g_Acc, Execute:= TRUE);
	IF DoMove.Busy THEN 
		iStatus:=iStatus + 1;
	END_IF
	
2: // Wait for Move Finish
	DoMove(Axis:=X, Distance:= g_PosDistance, Velocity:=g_Vel, Acceleration:=g_Acc, Deceleration:=g_Acc, Execute:= TRUE);
	IF DoMove.Done AND X.nAxisState=standstill THEN 
		DoMove(Axis:=X, Execute:= FALSE);
		iStatus:=iStatus + 1;
	END_IF
	
3: //Wait Time
	g_MoveDwellPos := TRUE;
	TimerON(PT:=tWait, IN:=TRUE);
	IF TimerON.Q=TRUE THEN
		TimerON(IN:=FALSE,PT:=T#0S);
		iStatus:=iStatus + 1;
		g_MoveDwellPos :=  FALSE;
	END_IF

4: //Start positive move
	DoMove(Axis:=X, Distance:= g_NegDistance, Velocity:=g_Vel, Acceleration:=g_Acc, Deceleration:=g_Acc, Execute:= TRUE);
	IF DoMove.Busy THEN 
		iStatus:=iStatus + 1;
	END_IF
	
5: // Wait for Move Finish
	DoMove(Axis:=X, Distance:= g_NegDistance, Velocity:=g_Vel, Acceleration:=g_Acc, Deceleration:=g_Acc, Execute:= TRUE);
	IF DoMove.Done AND X.nAxisState=standstill THEN 
		DoMove(Axis:=X, Execute:= FALSE);
		iStatus:=iStatus + 1;
	END_IF
	
6: //Wait Time
	g_MoveDwellNeg := TRUE;
	TimerON(PT:=tWait, IN:=TRUE);
	IF TimerON.Q=TRUE THEN
		TimerON(IN:=FALSE,PT:=T#0S);
		iStatus:=0;
		g_MoveDwellNeg := FALSE;
	END_IF

10: //IF DC Out of Sync
	EtherCAT_Master.xRestart := TRUE;
	EtherCAT_Master();
	TimerRecover(PT:=tWait, IN:=TRUE);
	IF TimerRecover.Q=TRUE THEN
		TimerRecover(IN:=FALSE,PT:=T#0S);
		iStatus:=11;
	END_IF
	
11: //Re Initialize Drive
	Restart_Axis(Axis:=X, bExecute:= TRUE);
	IF Restart_Axis.bDone THEN
		Restart_Axis(Axis:=X, bExecute:= FALSE);
		g_LostSync := FALSE;
		g_FirstSync := FALSE;
		iStatus := -2;
	END_IF
	
		
END_CASE;

END_PROGRAM

// POU_X
PROGRAM POU_X
VAR	
	ControlX : IO_AxisControl;
	X_Ready: BOOL;
END_VAR

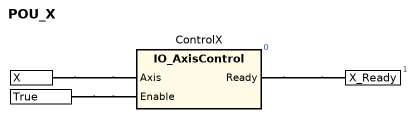
ControlX(Axis := X, Enable := True); // IO_AxisControl
X_Ready := ControlX.Ready;

END_PROGRAM

// InitSDO_Y
FUNCTION_BLOCK InitSDO_Y
VAR_IN_OUT
	Axis : AXIS_REF_ETC_SM3;
END_VAR
VAR_INPUT
	Execute:BOOL;
END_VAR
VAR_OUTPUT
	Done:BOOL;
	Busy:BOOL;
	Error: BOOL;
	
END_VAR
VAR
	SDOIndex:UINT:=8595;	//0x2193;
	SDOSubIndex:USINT:=0;
	numOutputs : USINT:=3;
	SDO_Write_OutConfig: SMC3_ETC_WriteParameter_CoE;
	iSubIndex: USINT;
END_VAR

numOutputs := 6;

FOR iSubIndex := 1 TO numOutputs DO
	WHILE (NOT(SDO_Write_OutConfig.xDone)) DO
		SDO_Write_OutConfig(uiIndex := SDOIndex, usiSubIndex := iSubIndex, usiDatalength := 2, dwValue := 2, Axis := Y, xExecute:= TRUE);	
	END_WHILE;
	SDO_Write_OutConfig(Axis := Y, xExecute:= FALSE);
END_FOR;

END_FUNCTION_BLOCK

// RunMotion_Y_old
PROGRAM RunMotion_Y_old
VAR
	AxisControl : IO_AxisControl;
	iStatus: INT := -2;
	DoMove : MC_MoveRelative;
	TimerON:TON;
	tWait : TIME := T#5S;
	tWaitPowerup: TIME := T#30S;
	ScanTimeMax: DINT;
	ScanTimeMin: DINT;
	Got_DC_OutOfSync: BOOL;

END_VAR

IF iStatus > -1 AND NOT(DC_InSync) THEN
	Got_DC_OutOfSync := TRUE;
END_IF

CASE iStatus OF
	
-2: //Wait Time
	//TimerON(PT:=tWaitPowerup, IN:=TRUE);
	IF EtherCAT_Master.xConfigFinished AND DC_InSync THEN
		//TimerON(IN:=FALSE,PT:=T#0S);
		iStatus:=iStatus + 1;
	END_IF
	
-1: //Wait Time
	AxisControl(Axis:=Y, Enable:=TRUE);
	IF DC_InSync THEN
		iStatus:=iStatus + 1;
	END_IF
	
	
0: //Wait for Drive to be ready
	AxisControl(Axis:=Y, Enable:=TRUE);
	//In_Power:=TRUE;
	IF AxisControl.Ready AND Y.nAxisState=standstill THEN
		iStatus:=iStatus + 1;	
	END_IF;
	
1: //Start positive move
	DoMove(Axis:=Y, Distance:= g_PosDistance, Velocity:=g_Vel, Acceleration:=g_Acc, Deceleration:=g_Acc, Execute:= TRUE);
	IF DoMove.Busy THEN 
		iStatus:=iStatus + 1;
	END_IF
	
2: // Wait for Move Finish
	DoMove(Axis:=Y, Distance:= g_PosDistance, Velocity:=g_Vel, Acceleration:=g_Acc, Deceleration:=g_Acc, Execute:= TRUE);
	IF DoMove.Done AND Y.nAxisState=standstill THEN 
		DoMove(Axis:=Y, Execute:= FALSE);
		iStatus:=iStatus + 1;
	END_IF
	
3: //Wait Time
	g_MoveDwellPos_Y := TRUE;
	TimerON(PT:=tWait, IN:=TRUE);
	IF TimerON.Q=TRUE THEN
		TimerON(IN:=FALSE,PT:=T#0S);
		iStatus:=iStatus + 1;
		g_MoveDwellPos_Y :=  FALSE;
	END_IF

4: //Start positive move
	DoMove(Axis:=Y, Distance:= g_NegDistance, Velocity:=g_Vel, Acceleration:=g_Acc, Deceleration:=g_Acc, Execute:= TRUE);
	IF DoMove.Busy THEN 
		iStatus:=iStatus + 1;
	END_IF
	
5: // Wait for Move Finish
	DoMove(Axis:=Y, Distance:= g_NegDistance, Velocity:=g_Vel, Acceleration:=g_Acc, Deceleration:=g_Acc, Execute:= TRUE);
	IF DoMove.Done AND Y.nAxisState=standstill THEN 
		DoMove(Axis:=Y, Execute:= FALSE);
		iStatus:=iStatus + 1;
	END_IF
	
6: //Wait Time
	g_MoveDwellNeg_Y := TRUE;
	TimerON(PT:=tWait, IN:=TRUE);
	IF TimerON.Q=TRUE THEN
		TimerON(IN:=FALSE,PT:=T#0S);
		iStatus:=0;
		g_MoveDwellNeg_Y := FALSE;
	END_IF

	
END_CASE;

END_PROGRAM

// RunSDO_Y
PROGRAM RunSDO_Y
VAR
	iStatus : INT := -2;
	GetPosition : GetSDO;
	ExpectedValue: REAL;
	ActualValue: DWORD;
	InitializeSDO: InitSDO_Y;
	ScanTimeMax: DINT;
	ScanTimeMin: DINT;
	DC_InSync: BOOL;
	Got_DC_OutOfSync: BOOL;

	InitalValue: DWORD;
END_VAR

EtherCAT_Master();
ScanTimeMax := EtherCAT_Master.m_master.m_diMaxSyncTime;
ScanTimeMin := EtherCAT_Master.m_master.m_diMinSyncTime;
DC_InSync := EtherCAT_Master.xDistributedClockInSync;

IF iStatus > -1 AND NOT(DC_InSync) THEN
	Got_DC_OutOfSync := TRUE;
END_IF

CASE iStatus OF
	
-2: //Initialize
	IF EtherCAT_Master.xConfigFinished AND DC_InSync THEN //AND RunMotion.AxisControl.Ready THEN
		InitializeSDO(Axis:= Y, Execute:= TRUE);
		GetPosition(Axis:=Y, Execute:=TRUE);
		iStatus:=iStatus + 1;
	END_IF

-1: //Wait for Init Finish
	InitializeSDO(Axis:= Y, Execute:= TRUE);
	GetPosition(Axis:=Y, Execute:=TRUE);
	IF GetPosition.Done THEN
		InitalValue := GetPosition.Position;
		GetPosition(Axis:=Y, Execute:=FALSE);
		
		IF InitializeSDO.Done THEN
			InitializeSDO(Axis:= Y, Execute:= FALSE);
			iStatus:=iStatus + 1;
		END_IF
	END_IF;
	

0 : //Wait for Dwell
	IF g_MoveDwellPos OR g_MoveDwellNeg THEN
		iStatus:=iStatus + 1;
	END_IF;
	
1 : //Call GetPosition
	GetPosition(Axis:=Y, Execute:=TRUE);
	iStatus:=iStatus + 1;
	RETURN;
	
2: //Wait for GetPosition to finish
	GetPosition(Axis:=Y, Execute:=TRUE);
	IF GetPosition.Done THEN
		ActualValue := GetPosition.Position;
		GetPosition(Axis:=Y, Execute:=FALSE);
		iStatus := iStatus + 1;
	END_IF;
	
3: //Check Position
	IF g_MoveDwellPos_Y THEN
		ExpectedValue := g_PosDistance * 4000 + InitalValue;
		g_GotSDO_Y_PostionPos := ActualValue < (ExpectedValue * 1.1) AND ActualValue > (ExpectedValue *0.9);
	END_IF;
	
	IF g_MoveDwellNeg_Y THEN
		ExpectedValue := g_PosDistance * 4000 + g_NegDistance * 4000 + InitalValue;
		g_GotSDO_Y_PostionNeg := ActualValue < (ExpectedValue * 1.1) AND ActualValue > (ExpectedValue *0.9);
	END_IF;
	iStatus := iStatus + 1;
	
4: //Wait for motion
	IF g_MoveDwellNeg_Y = FALSE AND g_MoveDwellPos_Y = FALSE  THEN
		iStatus := 0;
	END_IF;
	
END_CASE;

END_PROGRAM

// RunSDO_AOut_Y
PROGRAM RunSDO_AOut_Y
VAR
	iStatus: INT := -1;
	iCycle: INT;
	iCycleMin: INT := -10;
	iCycleMax: INT := 2460;
	DoOutputs : SetSDO_AOut_Y;
	DoInputs : GetSDO_AOut_Y;
	TimerON : TON;
	tWait: TIME := T#500ms;
	iIncrement: INT := 123;
	rExpectedValue: REAL;
	rActualValue: REAL;
//	cavConfig: ConfigAnalogVoltage;
	ResetError: BOOL;
	
	ValueMin1: REAL;
	ValueMax1: REAL;
	ValueMin2: REAL;
	ValueMax2: REAL;
	
	ScanTimeMax: DINT;
	ScanTimeMin: DINT;
	DC_InSync: BOOL;
	Got_DC_OutOfSync: BOOL;

	ExpectedValue1: INT;
	ExpectedValue2: INT;
	ActualValue1: INT;
	ActualValue2: INT;
	
	AOut1_Passed : BOOL;
	AOut2_Passed : BOOL;
	
END_VAR

EtherCAT_Master();
ScanTimeMax := EtherCAT_Master.m_master.m_diMaxSyncTime;
ScanTimeMin := EtherCAT_Master.m_master.m_diMinSyncTime;
DC_InSync := EtherCAT_Master.xDistributedClockInSync;

IF iStatus > -1 AND NOT(DC_InSync) THEN
	Got_DC_OutOfSync := TRUE;
END_IF

CASE iStatus OF
	
	
-1: //Wait for EtherCAT
	IF EtherCAT_Master.xConfigFinished  THEN
		iStatus:=iStatus + 1;
	END_IF
	
0: //Set Outputs
	ExpectedValue1 := 15000 + iCycle;
	ExpectedValue2 := 15000 - iCycle;
	
	DoOutputs(Axis:=Y, AOut1 := ExpectedValue1, AOut2 := ExpectedValue2, Execute:=TRUE);
	
	IF DoOutputs.Done THEN
		iCycle:=iCycle + iIncrement;
		IF iCycle >= iCycleMax THEN
			iCycle:=0;
		END_IF;
		iStatus := iStatus + 1;	
	END_IF
1: //Wait Time
	TimerON(PT:=tWait, IN:=TRUE);
	IF TimerON.Q=TRUE THEN
		TimerON(IN:=FALSE,PT:=T#0S);
		iStatus := iStatus + 1;
	END_IF
2: //Check Inputs
	DoInputs(Axis:=Y, Execute:=TRUE );
	
	IF DoInputs.Done = TRUE THEN
		ActualValue1:=DoInputs.AOut1;
		ActualValue2:=DoInputs.AOut2;
		
		ValueMin1:=ExpectedValue1 * 0.9;
		ValueMax1:=ExpectedValue1 * 1.1;
	
		ValueMin2:=ExpectedValue2 * 0.9;
		ValueMax2:=ExpectedValue2 * 1.1;
		
		AOut1_Passed := (ActualValue1 > ValueMin1) AND (ActualValue1 < ValueMax1);
		AOut2_Passed := (ActualValue2 > ValueMin2) AND (ActualValue2 < ValueMax2);
		
		iStatus := iStatus + 1;	
		DoOutputs(Axis := Y, Execute:=FALSE);
		DoInputs(Axis := Y, Execute:=FALSE);
	END_IF
3: //Wait Time
	TimerON(PT:=tWait, IN:=TRUE);
	IF TimerON.Q=TRUE THEN
		TimerON(IN:=FALSE,PT:=T#0S);
		iStatus:=0;
	END_IF
	

END_CASE;

END_PROGRAM

// SetSDO_AOut_Y
FUNCTION_BLOCK SetSDO_AOut_Y
VAR_IN_OUT
	Axis : AXIS_REF_ETC_SM3;
END_VAR
VAR_INPUT
	Execute:BOOL;
	AOut1: INT;
	AOut2: INT;
END_VAR
VAR_OUTPUT
	Done:BOOL;
	Busy:BOOL;
	Error: BOOL;
	
END_VAR
VAR
	AOut1_PosIndex:UINT:=8217;	//0x2019;
	AOut1_PosSubIndex:USINT:=0;
	AOut2_PosIndex:UINT:=8234;	//0x202A;
	AOut2_PosSubIndex:USINT:=0;
	
	SDO_Write_C3_AOut1: SMC3_ETC_WriteParameter_CoE;
	SDO_Write_C3_AOut2: SMC3_ETC_WriteParameter_CoE;
END_VAR
VAR // added by the converter: edge detectors and wires of the graphical bodies
    _w1 : ANY;
    _w2, _w3 : BOOL;
END_VAR

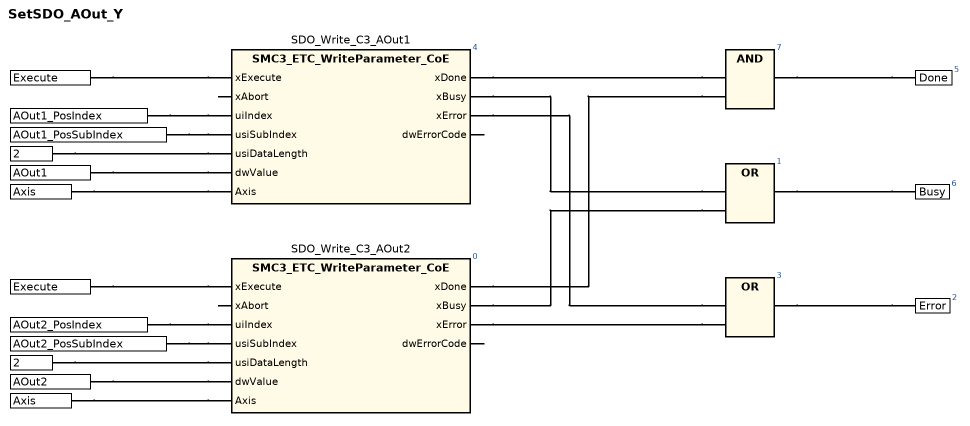
SDO_Write_C3_AOut2(
    xExecute := Execute,
    uiIndex := AOut2_PosIndex,
    usiSubIndex := AOut2_PosSubIndex,
    usiDataLength := 2,
    dwValue := AOut2,
    Axis := Axis); // SMC3_ETC_WriteParameter_CoE
_w1 := SDO_Write_C3_AOut1.xBusy OR SDO_Write_C3_AOut2.xBusy;
Error := _w2;
_w2 := SDO_Write_C3_AOut1.xError OR SDO_Write_C3_AOut2.xError;
SDO_Write_C3_AOut1(
    xExecute := Execute,
    uiIndex := AOut1_PosIndex,
    usiSubIndex := AOut1_PosSubIndex,
    usiDataLength := 2,
    dwValue := AOut1,
    Axis := Axis); // SMC3_ETC_WriteParameter_CoE
Done := _w3;
Busy := _w1;
_w3 := SDO_Write_C3_AOut1.xDone AND SDO_Write_C3_AOut2.xDone;

END_FUNCTION_BLOCK

// GetSDO_AOut_Y
FUNCTION_BLOCK GetSDO_AOut_Y
VAR_IN_OUT
	Axis : AXIS_REF_ETC_SM3;
END_VAR
VAR_INPUT
	Execute:BOOL;
END_VAR
VAR_OUTPUT
	Done:BOOL;
	Busy:BOOL;
	Error: BOOL;
	AOut1: INT;
	AOut2: INT;

END_VAR
VAR
	AOut1_PosIndex:UINT:=8217;	//0x2019;
	AOut1_PosSubIndex:USINT:=0;
	AOut2_PosIndex:UINT:=8234;	//0x202A;
	AOut2_PosSubIndex:USINT:=0;

	SDO_Read_C3_AOut1: SMC3_ETC_ReadParameter_CoE;
	SDO_Read_C3_AOut2: SMC3_ETC_ReadParameter_CoE;
END_VAR
VAR // added by the converter: edge detectors and wires of the graphical bodies
    _w1, _w2, _w3 : BOOL;
    _w4, _w5 : INT;
END_VAR

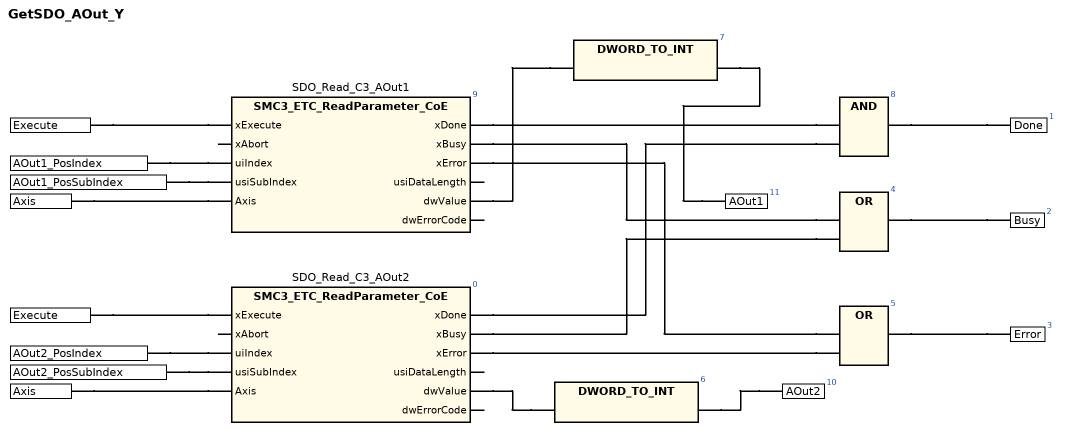
SDO_Read_C3_AOut2(
    xExecute := Execute,
    uiIndex := AOut2_PosIndex,
    usiSubIndex := AOut2_PosSubIndex,
    Axis := Axis); // SMC3_ETC_ReadParameter_CoE
Done := _w1;
Busy := _w2;
Error := _w3;
_w2 := SDO_Read_C3_AOut1.xBusy OR SDO_Read_C3_AOut2.xBusy;
_w3 := SDO_Read_C3_AOut1.xError OR SDO_Read_C3_AOut2.xError;
_w4 := DWORD_TO_INT(SDO_Read_C3_AOut2.dwValue);
_w5 := DWORD_TO_INT(SDO_Read_C3_AOut1.dwValue);
_w1 := SDO_Read_C3_AOut1.xDone AND SDO_Read_C3_AOut2.xDone;
SDO_Read_C3_AOut1(
    xExecute := Execute,
    uiIndex := AOut1_PosIndex,
    usiSubIndex := AOut1_PosSubIndex,
    Axis := Axis); // SMC3_ETC_ReadParameter_CoE
AOut2 := _w4;
AOut1 := _w5;

END_FUNCTION_BLOCK

// GetSDO_Y
FUNCTION_BLOCK GetSDO_Y
VAR_IN_OUT
	Axis : AXIS_REF_ETC_SM3;
END_VAR
VAR_INPUT
	Execute:BOOL;
END_VAR
VAR_OUTPUT
	Done:BOOL;
	Busy:BOOL;
	Error: BOOL;
	Position:DWORD;
	
END_VAR
VAR
	SDO_Read_C3_Position: SMC3_ETC_ReadParameter_CoE;
	PosIndex:UINT:=8768;
	PosSubIndex:USINT:=0;
END_VAR

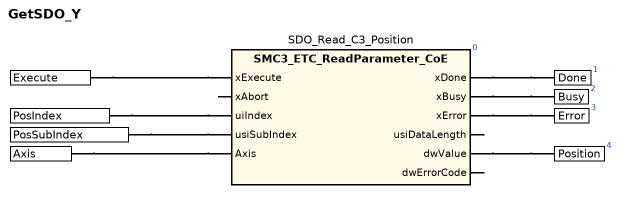
SDO_Read_C3_Position(xExecute := Execute, uiIndex := PosIndex, usiSubIndex := PosSubIndex, Axis := Axis); // SMC3_ETC_ReadParameter_CoE
Done := SDO_Read_C3_Position.xDone;
Busy := SDO_Read_C3_Position.xBusy;
Error := SDO_Read_C3_Position.xError;
Position := SDO_Read_C3_Position.dwValue;

END_FUNCTION_BLOCK

// RunMotion_Z_old
PROGRAM RunMotion_Z_old
VAR
	AxisControl : IO_AxisControl;
	iStatus: INT := -2;
	DoMove : MC_MoveRelative;
	TimerON:TON;
	tWait : TIME := T#5S;
	tWaitPowerup: TIME := T#30S;
	Got_DC_OutOfSync: BOOL;

	AxisVar: AXIS_REF_SM3;
END_VAR

AxisVar := Z;

IF iStatus > -1 AND NOT(DC_InSync) THEN
	Got_DC_OutOfSync := TRUE;
END_IF

CASE iStatus OF
	
-2: //Wait Time
	//TimerON(PT:=tWaitPowerup, IN:=TRUE);
	IF EtherCAT_Master.xConfigFinished AND DC_InSync THEN
		//TimerON(IN:=FALSE,PT:=T#0S);
		iStatus:=iStatus + 1;
	END_IF
	
-1: //Wait Time
	AxisControl(Axis:=Z, Enable:=TRUE);
	IF DC_InSync THEN
		iStatus:=iStatus + 1;
	END_IF
	
	
0: //Wait for Drive to be ready
	AxisControl(Axis:=Z, Enable:=TRUE);
	In_Power:=TRUE;
	IF AxisControl.Ready AND Z.nAxisState=standstill THEN
		iStatus:=iStatus + 1;	
	END_IF;
	
1: //Start positive move
	DoMove(Axis:=Z, Distance:= g_PosDistance, Velocity:=g_Vel, Acceleration:=g_Acc, Deceleration:=g_Acc, Execute:= TRUE);
	IF DoMove.Busy THEN 
		iStatus:=iStatus + 1;
	END_IF
	
2: // Wait for Move Finish
	DoMove(Axis:=Z, Distance:= g_PosDistance, Velocity:=g_Vel, Acceleration:=g_Acc, Deceleration:=g_Acc, Execute:= TRUE);
	IF DoMove.Done AND Z.nAxisState=standstill THEN 
		DoMove(Axis:=Z, Execute:= FALSE);
		iStatus:=iStatus + 1;
	END_IF
	
3: //Wait Time
	g_MoveDwellPos := TRUE;
	TimerON(PT:=tWait, IN:=TRUE);
	IF TimerON.Q=TRUE THEN
		TimerON(IN:=FALSE,PT:=T#0S);
		iStatus:=iStatus + 1;
		g_MoveDwellPos :=  FALSE;
	END_IF

4: //Start positive move
	DoMove(Axis:=Z, Distance:= g_NegDistance, Velocity:=g_Vel, Acceleration:=g_Acc, Deceleration:=g_Acc, Execute:= TRUE);
	IF DoMove.Busy THEN 
		iStatus:=iStatus + 1;
	END_IF
	
5: // Wait for Move Finish
	DoMove(Axis:=Z, Distance:= g_NegDistance, Velocity:=g_Vel, Acceleration:=g_Acc, Deceleration:=g_Acc, Execute:= TRUE);
	IF DoMove.Done AND Z.nAxisState=standstill THEN 
		DoMove(Axis:=Z, Execute:= FALSE);
		iStatus:=iStatus + 1;
	END_IF
	
6: //Wait Time
	g_MoveDwellNeg := TRUE;
	TimerON(PT:=tWait, IN:=TRUE);
	IF TimerON.Q=TRUE THEN
		TimerON(IN:=FALSE,PT:=T#0S);
		iStatus:=0;
		g_MoveDwellNeg := FALSE;
	END_IF

	
END_CASE;

END_PROGRAM

// RunMotion_A
PROGRAM RunMotion_A
VAR
	AxisControl : IO_AxisControl;
	iStatus: INT := -2;
	DoMove : MC_MoveRelative;
	TimerON:TON;
	tWait : TIME := T#5S;
	tWaitPowerup: TIME := T#30S;
	Got_DC_OutOfSync: BOOL;

	AxisVar: AXIS_REF_SM3;
END_VAR

AxisVar := A;

IF iStatus > -1 AND NOT(DC_InSync) THEN
	Got_DC_OutOfSync := TRUE;
END_IF

CASE iStatus OF
	
-2: //Wait Time
	//TimerON(PT:=tWaitPowerup, IN:=TRUE);
	IF EtherCAT_Master.xConfigFinished AND DC_InSync THEN
		//TimerON(IN:=FALSE,PT:=T#0S);
		iStatus:=iStatus + 1;
	END_IF
	
-1: //Wait Time
	AxisControl(Axis:=A, Enable:=TRUE);
	IF DC_InSync THEN
		iStatus:=iStatus + 1;
	END_IF
	
	
0: //Wait for Drive to be ready
	AxisControl(Axis:=A, Enable:=TRUE);
	In_Power:=TRUE;
	IF AxisControl.Ready AND A.nAxisState=standstill THEN
		iStatus:=iStatus + 1;	
	END_IF;
	
1: //Start positive move
	DoMove(Axis:=A, Distance:= g_PosDistance, Velocity:=g_Vel, Acceleration:=g_Acc, Deceleration:=g_Acc, Execute:= TRUE);
	IF DoMove.Busy THEN 
		iStatus:=iStatus + 1;
	END_IF
	
2: // Wait for Move Finish
	DoMove(Axis:=A, Distance:= g_PosDistance, Velocity:=g_Vel, Acceleration:=g_Acc, Deceleration:=g_Acc, Execute:= TRUE);
	IF DoMove.Done AND A.nAxisState=standstill THEN 
		DoMove(Axis:=A, Execute:= FALSE);
		iStatus:=iStatus + 1;
	END_IF
	
3: //Wait Time
	g_MoveDwellPos := TRUE;
	TimerON(PT:=tWait, IN:=TRUE);
	IF TimerON.Q=TRUE THEN
		TimerON(IN:=FALSE,PT:=T#0S);
		iStatus:=iStatus + 1;
		g_MoveDwellPos :=  FALSE;
	END_IF

4: //Start positive move
	DoMove(Axis:=A, Distance:= g_NegDistance, Velocity:=g_Vel, Acceleration:=g_Acc, Deceleration:=g_Acc, Execute:= TRUE);
	IF DoMove.Busy THEN 
		iStatus:=iStatus + 1;
	END_IF
	
5: // Wait for Move Finish
	DoMove(Axis:=A, Distance:= g_NegDistance, Velocity:=g_Vel, Acceleration:=g_Acc, Deceleration:=g_Acc, Execute:= TRUE);
	IF DoMove.Done AND A.nAxisState=standstill THEN 
		DoMove(Axis:=A, Execute:= FALSE);
		iStatus:=iStatus + 1;
	END_IF
	
6: //Wait Time
	g_MoveDwellNeg := TRUE;
	TimerON(PT:=tWait, IN:=TRUE);
	IF TimerON.Q=TRUE THEN
		TimerON(IN:=FALSE,PT:=T#0S);
		iStatus:=0;
		g_MoveDwellNeg := FALSE;
	END_IF

	
END_CASE;

END_PROGRAM

// AllTaskInfo
FUNCTION AllTaskInfo : ARRAY[1..20] OF Task_Info2
VAR_INPUT
END_VAR
VAR
	hTask 	: RTS_IEC_HANDLE; (* task handle *)
	iTasks  : INT; (* task counter *)
	pTask 	: POINTER TO Task_Info2; (* pointer to task information *)
	sAppName: STRING := 'Application'; (* name of the application *)
	Result	: RTS_IEC_RESULT; (* error code *)
END_VAR

(* Information of all tasks are stored in an array. *)
iTasks   := 0;
hTask := IecTaskGetFirst(pszAppName:=ADR(sAppName), pResult:=ADR(Result));
WHILE hTask <> RTS_INVALID_HANDLE AND Result = 0 DO
	iTasks   := iTasks + 1;
	pTask    := IecTaskGetInfo2(hIecTask:=hTask, pResult:=ADR(Result));
	IF pTask <> 0 AND Result = 0 THEN
		AllTaskInfo[iTasks] := pTask^;
	END_IF
	
	(* Get the next task *)
	hTask := IecTaskGetNext(pszAppName:=ADR(sAppName), hPrevIecTask:=hTask, pResult:=ADR(Result));
END_WHILE

END_FUNCTION

// RunMotion_Y
PROGRAM RunMotion_Y
VAR
	AxisControl : IO_AxisControl;
	iStatus: INT := -2;
	DoMove : MC_MoveRelative;
	TimerON:TON;
	tWait : TIME := T#5S;
	tWaitPowerup: TIME := T#30S;
	Got_DC_OutOfSync: BOOL;
	EnableAxisControl: BOOL := FALSE;
	HMI_ActualPosition : INT;
	
	
	

	AxisVar: AXIS_REF_SM3;
	Restart_Axis : SMC3_ReinitDrive;
	TimerRecover : TON;
	ActualPositionY: LREAL;
END_VAR

AxisVar := Y;

IF iStatus > -1 AND NOT(DC_InSync) THEN
	Got_DC_OutOfSync := TRUE;
//  Commented out the recovery mechanism to trap the error	
//	iStatus := 10; 
END_IF

CASE iStatus OF
	
-2: //Wait Time
	EnableAxisControl:= FALSE;
	
	//TimerON(PT:=tWaitPowerup, IN:=TRUE);
	IF EtherCAT_Master.xConfigFinished AND DC_InSync THEN
		//TimerON(IN:=FALSE,PT:=T#0S);
		iStatus:=iStatus + 1;
	END_IF
	
-1: //Wait Time
	EnableAxisControl:=TRUE;
	
	IF DC_InSync THEN
		iStatus:=iStatus + 1;
	END_IF
	
	
0: //Wait for Drive to be ready
	//AxisControl(Axis:=X, Enable:=TRUE);
	//In_Power:=TRUE;
	IF AxisControl.Ready AND Y.nAxisState=standstill THEN
		IF In_Cycle = TRUE THEN
			iStatus:=iStatus + 1;
		ELSE
			iStatus:=0;	
		END_IF
	END_IF;
	
1: //Start positive move
	DoMove(Axis:=Y, Distance:= g_PosDistance, Velocity:=g_Vel, Acceleration:=g_Acc, Deceleration:=g_Acc, Execute:= TRUE);
	IF DoMove.Busy THEN 
		IF In_Cycle = TRUE THEN
			iStatus:=iStatus + 1;
		ELSE
			iStatus:=0;	
		END_IF
	END_IF
	
2: // Wait for Move Finish
	DoMove(Axis:=Y, Distance:= g_PosDistance, Velocity:=g_Vel, Acceleration:=g_Acc, Deceleration:=g_Acc, Execute:= TRUE);
	IF DoMove.Done AND Y.nAxisState=standstill THEN 
		DoMove(Axis:=Y, Execute:= FALSE);
		
		IF In_Cycle = TRUE THEN
			iStatus:=iStatus + 1;
		ELSE
			iStatus:=0;	
		END_IF
	END_IF
	
3: //Wait Time
	g_MoveDwellPos := TRUE;
	TimerON(PT:=tWait, IN:=TRUE);
	IF TimerON.Q=TRUE THEN
		TimerON(IN:=FALSE,PT:=T#0S);
		g_MoveDwellPos :=  FALSE;
		
		IF In_Cycle = TRUE THEN
			iStatus:=iStatus + 1;
		ELSE
			iStatus:=0;	
		END_IF
		
	END_IF

4: //Start negative move
	DoMove(Axis:=Y, Distance:= g_NegDistance, Velocity:=g_Vel, Acceleration:=g_Acc, Deceleration:=g_Acc, Execute:= TRUE);
	IF DoMove.Busy THEN 
		IF In_Cycle = TRUE THEN
			iStatus:=iStatus + 1;
		ELSE
			iStatus:=0;	
		END_IF
	END_IF
	
5: // Wait for Move Finish
	DoMove(Axis:=Y, Distance:= g_NegDistance, Velocity:=g_Vel, Acceleration:=g_Acc, Deceleration:=g_Acc, Execute:= TRUE);
	IF DoMove.Done AND Y.nAxisState=standstill THEN 
		DoMove(Axis:=Y, Execute:= FALSE);
		IF In_Cycle = TRUE THEN
			iStatus:=iStatus + 1;
		ELSE
			iStatus:=0;	
		END_IF
	END_IF
	
6: //Wait Time
	g_MoveDwellNeg := TRUE;
	TimerON(PT:=tWait, IN:=TRUE);
	IF TimerON.Q=TRUE THEN
		TimerON(IN:=FALSE,PT:=T#0S);
		g_MoveDwellNeg := FALSE;
		IF In_Cycle = TRUE THEN
			iStatus:= 1;
		ELSE
			iStatus:=0;	
		END_IF
	END_IF

10: //IF DC Out of Sync
	EnableAxisControl:= FALSE;
	EtherCAT_Master.xRestart := TRUE;
	EtherCAT_Master();
	TimerRecover(PT:=tWait, IN:=TRUE);
	IF TimerRecover.Q=TRUE THEN
		TimerRecover(IN:=FALSE,PT:=T#0S);
		iStatus:=11;
	END_IF
	
11: //Re Initialize Drive
	Restart_Axis(Axis:=Y, bExecute:= TRUE);
	IF Restart_Axis.bDone THEN
		Restart_Axis(Axis:=Y, bExecute:= FALSE);
		g_LostSync := FALSE;
		g_FirstSync := FALSE;
		iStatus := -2;
	END_IF
	
		
END_CASE;

AxisControl(Axis:=Y, Enable:=EnableAxisControl);
ActualPositionY:=AxisControl.Actual_Position;
HMI_ActualPosition := LREAL_TO_INT(ActualPositionY * 1000);

END_PROGRAM

// RunMotion_Z
PROGRAM RunMotion_Z
VAR
	AxisControl : IO_AxisControl;
	iStatus: INT := -2;
	DoMove : MC_MoveRelative;
	TimerON:TON;
	tWait : TIME := T#5S;
	tWaitPowerup: TIME := T#30S;
	Got_DC_OutOfSync: BOOL;
	EnableAxisControl: BOOL := FALSE;
	HMI_ActualPosition : INT;
	
	
	

	AxisVar: AXIS_REF_SM3;
	Restart_Axis : SMC3_ReinitDrive;
	TimerRecover : TON;
	ActualPositionZ: LREAL;
END_VAR

AxisVar := Z;

IF iStatus > -1 AND NOT(DC_InSync) THEN
	Got_DC_OutOfSync := TRUE;
//  Commented out the recovery mechanism to trap the error	
//	iStatus := 10; 
END_IF

CASE iStatus OF
	
-2: //Wait Time
	EnableAxisControl:= FALSE;
	
	//TimerON(PT:=tWaitPowerup, IN:=TRUE);
	IF EtherCAT_Master.xConfigFinished AND DC_InSync THEN
		//TimerON(IN:=FALSE,PT:=T#0S);
		iStatus:=iStatus + 1;
	END_IF
	
-1: //Wait Time
	EnableAxisControl:=TRUE;
	
	IF DC_InSync THEN
		iStatus:=iStatus + 1;
	END_IF
	
	
0: //Wait for Drive to be ready
	//AxisControl(Axis:=X, Enable:=TRUE);
	//In_Power:=TRUE;
	IF AxisControl.Ready AND Z.nAxisState=standstill THEN
		IF In_Cycle = TRUE THEN
			iStatus:=iStatus + 1;
		ELSE
			iStatus:=0;	
		END_IF
	END_IF;
	
1: //Start positive move
	DoMove(Axis:=Z, Distance:= g_PosDistance, Velocity:=g_Vel, Acceleration:=g_Acc, Deceleration:=g_Acc, Execute:= TRUE);
	IF DoMove.Busy THEN 
		IF In_Cycle = TRUE THEN
			iStatus:=iStatus + 1;
		ELSE
			iStatus:=0;	
		END_IF
	END_IF
	
2: // Wait for Move Finish
	DoMove(Axis:=Z, Distance:= g_PosDistance, Velocity:=g_Vel, Acceleration:=g_Acc, Deceleration:=g_Acc, Execute:= TRUE);
	IF DoMove.Done AND Z.nAxisState=standstill THEN 
		DoMove(Axis:=Z, Execute:= FALSE);
		
		IF In_Cycle = TRUE THEN
			iStatus:=iStatus + 1;
		ELSE
			iStatus:=0;	
		END_IF
	END_IF
	
3: //Wait Time
	g_MoveDwellPos := TRUE;
	TimerON(PT:=tWait, IN:=TRUE);
	IF TimerON.Q=TRUE THEN
		TimerON(IN:=FALSE,PT:=T#0S);
		g_MoveDwellPos :=  FALSE;
		
		IF In_Cycle = TRUE THEN
			iStatus:=iStatus + 1;
		ELSE
			iStatus:=0;	
		END_IF
		
	END_IF

4: //Start negative move
	DoMove(Axis:=Z, Distance:= g_NegDistance, Velocity:=g_Vel, Acceleration:=g_Acc, Deceleration:=g_Acc, Execute:= TRUE);
	IF DoMove.Busy THEN 
		IF In_Cycle = TRUE THEN
			iStatus:=iStatus + 1;
		ELSE
			iStatus:=0;	
		END_IF
	END_IF
	
5: // Wait for Move Finish
	DoMove(Axis:=Z, Distance:= g_NegDistance, Velocity:=g_Vel, Acceleration:=g_Acc, Deceleration:=g_Acc, Execute:= TRUE);
	IF DoMove.Done AND Z.nAxisState=standstill THEN 
		DoMove(Axis:=Z, Execute:= FALSE);
		IF In_Cycle = TRUE THEN
			iStatus:=iStatus + 1;
		ELSE
			iStatus:=0;	
		END_IF
	END_IF
	
6: //Wait Time
	g_MoveDwellNeg := TRUE;
	TimerON(PT:=tWait, IN:=TRUE);
	IF TimerON.Q=TRUE THEN
		TimerON(IN:=FALSE,PT:=T#0S);
		g_MoveDwellNeg := FALSE;
		IF In_Cycle = TRUE THEN
			iStatus:= 1;
		ELSE
			iStatus:=0;	
		END_IF
	END_IF

10: //IF DC Out of Sync
	EnableAxisControl:= FALSE;
	EtherCAT_Master.xRestart := TRUE;
	EtherCAT_Master();
	TimerRecover(PT:=tWait, IN:=TRUE);
	IF TimerRecover.Q=TRUE THEN
		TimerRecover(IN:=FALSE,PT:=T#0S);
		iStatus:=11;
	END_IF
	
11: //Re Initialize Drive
	Restart_Axis(Axis:=Z, bExecute:= TRUE);
	IF Restart_Axis.bDone THEN
		Restart_Axis(Axis:=Z, bExecute:= FALSE);
		g_LostSync := FALSE;
		g_FirstSync := FALSE;
		iStatus := -2;
	END_IF
	
		
END_CASE;

AxisControl(Axis:=Z, Enable:=EnableAxisControl);
ActualPositionZ:=AxisControl.Actual_Position;
HMI_ActualPosition := LREAL_TO_INT(ActualPositionZ * 1000);

END_PROGRAM

// GetTimeStampString_1
FUNCTION GetTimeStampString_1 : String
VAR_INPUT
END_VAR
VAR
	TimeStamp : SysTime;
	StructTimeStamp : SysTimeDate;
	Result : RTS_IEC_RESULT;
	StrDate : STRING;
	StrTime : STRING;
	
END_VAR

Result := systimertc.SysTimeRtcHighResGet(pTimestamp := TimeStamp);

Result := systimertc.SysTimeRtcConvertHighResToLocal(pTimeStamp:=TimeStamp, pDate:=StructTimeStamp);

StrDate := UINT_TO_STRING(StructTimeStamp.wYear);
IF StructTimeStamp.wMonth < 10 THEN 
	StrDate := Concat(Concat(StrDate, '0') , UINT_TO_STRING(StructTimeStamp.wMonth));
ELSE
	StrDate := Concat(StrDate , UINT_TO_STRING(StructTimeStamp.wMonth));
END_IF

IF StructTimeStamp.wDay < 10 THEN 
	StrDate := Concat(Concat(StrDate , '0') , UINT_TO_STRING(StructTimeStamp.wDay));
ELSE
	StrDate := Concat(StrDate , UINT_TO_STRING(StructTimeStamp.wDay));
END_IF


IF StructTimeStamp.wHour < 10 THEN 
	StrTime := Concat(Concat('0' , UINT_TO_STRING(StructTimeStamp.wHour)) , ':');
ELSE
	StrTime := Concat(UINT_TO_STRING(StructTimeStamp.wHour) , ':');
END_IF

IF StructTimeStamp.wMinute < 10 THEN 
	StrTime := Concat(Concat(Concat(StrTime , '0') , UINT_TO_STRING(StructTimeStamp.wMinute)), ':');
ELSE
	StrTime := Concat(Concat(StrTime , UINT_TO_STRING(StructTimeStamp.wMinute)), ':');
END_IF

IF StructTimeStamp.wSecond < 10 THEN 
	StrTime := Concat(Concat(Concat(StrTime , '0') , UINT_TO_STRING(StructTimeStamp.wSecond)) , '.');
ELSE
	StrTime := Concat(Concat(StrTime , UINT_TO_STRING(StructTimeStamp.wSecond)) , '.');
END_IF

IF StructTimeStamp.wMilliseconds < 10 THEN 
	StrTime := Concat(Concat(StrTime , '00') , UINT_TO_STRING(StructTimeStamp.wMilliseconds));
ELSE
	IF StructTimeStamp.wMilliseconds < 100 THEN 
		StrTime := Concat(Concat(StrTime , '0') , UINT_TO_STRING(StructTimeStamp.wMilliseconds));
	ELSE
		StrTime := Concat(StrTime , UINT_TO_STRING(StructTimeStamp.wMilliseconds));
	END_IF
END_IF

//GetTimeStampString := Concat(Concat(strDate , '-'), strTime);
GetTimeStampString := strTime;

END_FUNCTION
